(* IEC 61131-3 sources: elnaProjects/ElpcLogic/PomarKc7Unchanged/build_USO_ecl (part 3) *)

  (********************************************* Модуль A1-6 ******************************************************)

  AI_T_opornogo_podshipnika_nagnetatelia_t1_HA	:= ai.T_opornogo_podshipnika_nagnetatelia_t1.HA;
  AI_T_opornogo_podshipnika_nagnetatelia_t1_HL	:= ai.T_opornogo_podshipnika_nagnetatelia_t1.HL;
  AI_T_opornogo_podshipnika_nagnetatelia_t1_HW	:= ai.T_opornogo_podshipnika_nagnetatelia_t1.HW;
  AI_T_opornogo_podshipnika_nagnetatelia_t1_LL	:= ai.T_opornogo_podshipnika_nagnetatelia_t1.LL;
  AI_T_opornogo_podshipnika_nagnetatelia_t1_status := DWORD_TO_UDINT(ai.T_opornogo_podshipnika_nagnetatelia_t1.status);
  AI_T_opornogo_podshipnika_nagnetatelia_t1_value := ai.T_opornogo_podshipnika_nagnetatelia_t1.value;

  AI_T_opornogo_podshipnika_nagnetatelia_t2_HA	:= ai.T_opornogo_podshipnika_nagnetatelia_t2.HA;
  AI_T_opornogo_podshipnika_nagnetatelia_t2_HL	:= ai.T_opornogo_podshipnika_nagnetatelia_t2.HL;
  AI_T_opornogo_podshipnika_nagnetatelia_t2_HW	:= ai.T_opornogo_podshipnika_nagnetatelia_t2.HW;
  AI_T_opornogo_podshipnika_nagnetatelia_t2_LL	:= ai.T_opornogo_podshipnika_nagnetatelia_t2.LL;
  AI_T_opornogo_podshipnika_nagnetatelia_t2_status := DWORD_TO_UDINT(ai.T_opornogo_podshipnika_nagnetatelia_t2.status);
  AI_T_opornogo_podshipnika_nagnetatelia_t2_value := ai.T_opornogo_podshipnika_nagnetatelia_t2.value;

  AI_T_opornogo_podshipnika_nagnetatelia_t3_HA	:= ai.T_opornogo_podshipnika_nagnetatelia_t3.HA;
  AI_T_opornogo_podshipnika_nagnetatelia_t3_HL	:= ai.T_opornogo_podshipnika_nagnetatelia_t3.HL;
  AI_T_opornogo_podshipnika_nagnetatelia_t3_HW	:= ai.T_opornogo_podshipnika_nagnetatelia_t3.HW;
  AI_T_opornogo_podshipnika_nagnetatelia_t3_LL	:= ai.T_opornogo_podshipnika_nagnetatelia_t3.LL;
  AI_T_opornogo_podshipnika_nagnetatelia_t3_status := DWORD_TO_UDINT(ai.T_opornogo_podshipnika_nagnetatelia_t3.status);
  AI_T_opornogo_podshipnika_nagnetatelia_t3_value := ai.T_opornogo_podshipnika_nagnetatelia_t3.value;

  AI_T_oporno_upornogo_podshipnika_nagnetatelia_t4_HA	:= ai.T_oporno_upornogo_podshipnika_nagnetatelia_t4.HA;
  AI_T_oporno_upornogo_podshipnika_nagnetatelia_t4_HL	:= ai.T_oporno_upornogo_podshipnika_nagnetatelia_t4.HL;
  AI_T_oporno_upornogo_podshipnika_nagnetatelia_t4_HW	:= ai.T_oporno_upornogo_podshipnika_nagnetatelia_t4.HW;
  AI_T_oporno_upornogo_podshipnika_nagnetatelia_t4_LL	:= ai.T_oporno_upornogo_podshipnika_nagnetatelia_t4.LL;
  AI_T_oporno_upornogo_podshipnika_nagnetatelia_t4_status := DWORD_TO_UDINT(ai.T_oporno_upornogo_podshipnika_nagnetatelia_t4.status);
  AI_T_oporno_upornogo_podshipnika_nagnetatelia_t4_value := ai.T_oporno_upornogo_podshipnika_nagnetatelia_t4.value;

  AI_T_masla_do_AVOM_HL	:= ai.T_masla_do_AVOM.HL;
  AI_T_masla_do_AVOM_LL	:= ai.T_masla_do_AVOM.LL;
  AI_T_masla_do_AVOM_status := DWORD_TO_UDINT(ai.T_masla_do_AVOM.status);
  AI_T_masla_do_AVOM_value := ai.T_masla_do_AVOM.value;

  AI_T_masla_posle_AVOM_HL	:= ai.T_masla_posle_AVOM.HL;
  AI_T_masla_posle_AVOM_LL	:= ai.T_masla_posle_AVOM.LL;
  AI_T_masla_posle_AVOM_status := DWORD_TO_UDINT(ai.T_masla_posle_AVOM.status);
  AI_T_masla_posle_AVOM_value := ai.T_masla_posle_AVOM.value;

  AI_T_gaz_in_nagnetatelia_HL	          := ai.T_gaz_in_nagnetatelia.HL;
  AI_T_gaz_in_nagnetatelia_LL	          := ai.T_gaz_in_nagnetatelia.LL;
  AI_T_gaz_in_nagnetatelia_status := DWORD_TO_UDINT(ai.T_gaz_in_nagnetatelia.status);
  AI_T_gaz_in_nagnetatelia_value := ai.T_gaz_in_nagnetatelia.value;

  AI_T_gaz_out_nagnetatelia_HA	          := ai.T_gaz_out_nagnetatelia.HA;
  AI_T_gaz_out_nagnetatelia_HL	          := ai.T_gaz_out_nagnetatelia.HL;
  AI_T_gaz_out_nagnetatelia_HW	          := ai.T_gaz_out_nagnetatelia.HW;
  AI_T_gaz_out_nagnetatelia_LL	          := ai.T_gaz_out_nagnetatelia.LL;
  AI_T_gaz_out_nagnetatelia_status := DWORD_TO_UDINT(ai.T_gaz_out_nagnetatelia.status);
  AI_T_gaz_out_nagnetatelia_value := ai.T_gaz_out_nagnetatelia.value;

  (********************************************* Модуль A1-7 ******************************************************)

  AI_T_clodAir_dvigatelia_t1_HL	          := ai.T_clodAir_dvigatelia_t1.HL;
  AI_T_clodAir_dvigatelia_t1_LL	          := ai.T_clodAir_dvigatelia_t1.LL;
  AI_T_clodAir_dvigatelia_t1_status := DWORD_TO_UDINT(ai.T_clodAir_dvigatelia_t1.status);
  AI_T_clodAir_dvigatelia_t1_value := ai.T_clodAir_dvigatelia_t1.value;

  AI_T_hotAir_dvigatelia_t1_HL	          := ai.T_hotAir_dvigatelia_t1.HL;
  AI_T_hotAir_dvigatelia_t1_LL	          := ai.T_hotAir_dvigatelia_t1.LL;
  AI_T_hotAir_dvigatelia_t1_status := DWORD_TO_UDINT(ai.T_hotAir_dvigatelia_t1.status);
  AI_T_hotAir_dvigatelia_t1_value := ai.T_hotAir_dvigatelia_t1.value;

  (********************************************* Модуль A1-8 ******************************************************)

  AI_dPmaslo_gaz_HL	          := ai.dPmaslo_gaz.HL;
  AI_dPmaslo_gaz_LA	          := ai.dPmaslo_gaz.LA;
  AI_dPmaslo_gaz_LL	          := ai.dPmaslo_gaz.LL;
  AI_dPmaslo_gaz_LW	          := ai.dPmaslo_gaz.LW;
  AI_dPmaslo_gaz_MaxChangeUP	          := ai.dPmaslo_gaz.MaxChangeSpeed;
  AI_dPmaslo_gaz_MaxChangeDown	          := ai.dPmaslo_gaz.MaxChangeSpeedDown;
  AI_dPmaslo_gaz_status := DWORD_TO_UDINT(ai.dPmaslo_gaz.status);
  AI_dPmaslo_gaz_value := ai.dPmaslo_gaz.value;

  AI_dP_gaza_na_konfuzore_nagnetatelia_HL	          := ai.dP_gaza_na_konfuzore_nagnetatelia.HL;
  AI_dP_gaza_na_konfuzore_nagnetatelia_LL	          := ai.dP_gaza_na_konfuzore_nagnetatelia.LL;
  AI_dP_gaza_na_konfuzore_nagnetatelia_status := DWORD_TO_UDINT(ai.dP_gaza_na_konfuzore_nagnetatelia.status);
  AI_dP_gaza_na_konfuzore_nagnetatelia_value := ai.dP_gaza_na_konfuzore_nagnetatelia.value;

  AI_P_masla_uplotneniia_HL	:= ai.P_masla_uplotneniia.HL;
  AI_P_masla_uplotneniia_LL	:= ai.P_masla_uplotneniia.LL;
  AI_P_masla_uplotneniia_status := DWORD_TO_UDINT(ai.P_masla_uplotneniia.status);
  AI_P_masla_uplotneniia_value := ai.P_masla_uplotneniia.value;

  AI_P_gaza_na_vkhode_nagnetatelia_HL	:= ai.P_gaza_na_vkhode_nagnetatelia.HL;
  AI_P_gaza_na_vkhode_nagnetatelia_LL	:= ai.P_gaza_na_vkhode_nagnetatelia.LL;
  AI_P_gaza_na_vkhode_nagnetatelia_status := DWORD_TO_UDINT(ai.P_gaza_na_vkhode_nagnetatelia.status);
  AI_P_gaza_na_vkhode_nagnetatelia_value := ai.P_gaza_na_vkhode_nagnetatelia.value;

  AI_P_gaza_na_vykhode_nagnetatelia_HL	:= ai.P_gaza_na_vykhode_nagnetatelia.HL;
  AI_P_gaza_na_vykhode_nagnetatelia_LL	:= ai.P_gaza_na_vykhode_nagnetatelia.LL;
  AI_P_gaza_na_vykhode_nagnetatelia_status := DWORD_TO_UDINT(ai.P_gaza_na_vykhode_nagnetatelia.status);
  AI_P_gaza_na_vykhode_nagnetatelia_value := ai.P_gaza_na_vykhode_nagnetatelia.value;

  AI_P_masla_smazki_nizkoe_HL	          := ai.P_masla_smazki_nizkoe.HL;
  AI_P_masla_smazki_nizkoe_LA	          := ai.P_masla_smazki_nizkoe.LA;
  AI_P_masla_smazki_nizkoe_LL	          := ai.P_masla_smazki_nizkoe.LL;
  AI_P_masla_smazki_nizkoe_LW	          := ai.P_masla_smazki_nizkoe.LW;
  AI_P_masla_smazki_nizkoe_status := DWORD_TO_UDINT(ai.P_masla_smazki_nizkoe.status);
  AI_P_masla_smazki_nizkoe_value := ai.P_masla_smazki_nizkoe.value;

  AI_P_masla_smazki_srednee_posle_nasosov_HL	:= ai.P_masla_smazki_srednee_posle_nasosov.HL;
  AI_P_masla_smazki_srednee_posle_nasosov_LL	:= ai.P_masla_smazki_srednee_posle_nasosov.LL;
  AI_P_masla_smazki_srednee_posle_nasosov_LW	:= ai.P_masla_smazki_srednee_posle_nasosov.LW;
  AI_P_masla_smazki_srednee_posle_nasosov_status := DWORD_TO_UDINT(ai.P_masla_smazki_srednee_posle_nasosov.status);
  AI_P_masla_smazki_srednee_posle_nasosov_value := ai.P_masla_smazki_srednee_posle_nasosov.value;

  (********************************************* Модуль A1-9 ******************************************************)

  AI_Vibratciia_STD_t1_HA	:= ai.Vibratciia_STD_t1.HA;
  AI_Vibratciia_STD_t1_HL	:= ai.Vibratciia_STD_t1.HL;
  AI_Vibratciia_STD_t1_HW	:= ai.Vibratciia_STD_t1.HW;
  AI_Vibratciia_STD_t1_LL	:= ai.Vibratciia_STD_t1.LL;
  AI_Vibratciia_STD_t1_status := DWORD_TO_UDINT(ai.Vibratciia_STD_t1.status);
  AI_Vibratciia_STD_t1_value := ai.Vibratciia_STD_t1.value;

  AI_Vibratciia_STD_t2_HA	:= ai.Vibratciia_STD_t2.HA;
  AI_Vibratciia_STD_t2_HL	:= ai.Vibratciia_STD_t2.HL;
  AI_Vibratciia_STD_t2_HW	:= ai.Vibratciia_STD_t2.HW;
  AI_Vibratciia_STD_t2_LL	:= ai.Vibratciia_STD_t2.LL;
  AI_Vibratciia_STD_t2_status := DWORD_TO_UDINT(ai.Vibratciia_STD_t2.status);
  AI_Vibratciia_STD_t2_value := ai.Vibratciia_STD_t2.value;

  AI_Vibratciia_rotora_nagnetatelia_t1_HA	          := ai.Vibratciia_rotora_nagnetatelia_t1.HA;
  AI_Vibratciia_rotora_nagnetatelia_t1_HL	          := ai.Vibratciia_rotora_nagnetatelia_t1.HL;
  AI_Vibratciia_rotora_nagnetatelia_t1_HW	          := ai.Vibratciia_rotora_nagnetatelia_t1.HW;
  AI_Vibratciia_rotora_nagnetatelia_t1_LL	          := ai.Vibratciia_rotora_nagnetatelia_t1.LL;
  AI_Vibratciia_rotora_nagnetatelia_t1_status := DWORD_TO_UDINT(ai.Vibratciia_rotora_nagnetatelia_t1.status);
  AI_Vibratciia_rotora_nagnetatelia_t1_value := ai.Vibratciia_rotora_nagnetatelia_t1.value;

  AI_Vibratciia_rotora_nagnetatelia_t2_HA	          := ai.Vibratciia_rotora_nagnetatelia_t2.HA;
  AI_Vibratciia_rotora_nagnetatelia_t2_HL        	:= ai.Vibratciia_rotora_nagnetatelia_t2.HL;
  AI_Vibratciia_rotora_nagnetatelia_t2_HW    	:= ai.Vibratciia_rotora_nagnetatelia_t2.HW;
  AI_Vibratciia_rotora_nagnetatelia_t2_LL    	:= ai.Vibratciia_rotora_nagnetatelia_t2.LL;
  AI_Vibratciia_rotora_nagnetatelia_t2_status := DWORD_TO_UDINT(ai.Vibratciia_rotora_nagnetatelia_t2.status);
  AI_Vibratciia_rotora_nagnetatelia_t2_value := ai.Vibratciia_rotora_nagnetatelia_t2.value;

  AI_Vibratciia_rotora_nagnetatelia_t3_HA    	:= ai.Vibratciia_rotora_nagnetatelia_t3.HA;
  AI_Vibratciia_rotora_nagnetatelia_t3_HL    	:= ai.Vibratciia_rotora_nagnetatelia_t3.HL;
  AI_Vibratciia_rotora_nagnetatelia_t3_HW    	:= ai.Vibratciia_rotora_nagnetatelia_t3.HW;
  AI_Vibratciia_rotora_nagnetatelia_t3_LL    	:= ai.Vibratciia_rotora_nagnetatelia_t3.LL;
  AI_Vibratciia_rotora_nagnetatelia_t3_status := DWORD_TO_UDINT(ai.Vibratciia_rotora_nagnetatelia_t3.status);
  AI_Vibratciia_rotora_nagnetatelia_t3_value := ai.Vibratciia_rotora_nagnetatelia_t3.value;

  AI_Vibratciia_rotora_nagnetatelia_t4_HA    	:= ai.Vibratciia_rotora_nagnetatelia_t4.HA;
  AI_Vibratciia_rotora_nagnetatelia_t4_HL    	:= ai.Vibratciia_rotora_nagnetatelia_t4.HL;
  AI_Vibratciia_rotora_nagnetatelia_t4_HW    	:= ai.Vibratciia_rotora_nagnetatelia_t4.HW;
  AI_Vibratciia_rotora_nagnetatelia_t4_LL    	:= ai.Vibratciia_rotora_nagnetatelia_t4.LL;
  AI_Vibratciia_rotora_nagnetatelia_t4_status := DWORD_TO_UDINT(ai.Vibratciia_rotora_nagnetatelia_t4.status);
  AI_Vibratciia_rotora_nagnetatelia_t4_value := ai.Vibratciia_rotora_nagnetatelia_t4.value;

  AI_Osevoi_sdvig_rotora_nagnetatelia_HA    	:= ai.Osevoi_sdvig_rotora_nagnetatelia.HA;
  AI_Osevoi_sdvig_rotora_nagnetatelia_HL    	:= ai.Osevoi_sdvig_rotora_nagnetatelia.HL;
  AI_Osevoi_sdvig_rotora_nagnetatelia_HW    	:= ai.Osevoi_sdvig_rotora_nagnetatelia.HW;
  AI_Osevoi_sdvig_rotora_nagnetatelia_LA    	:= ai.Osevoi_sdvig_rotora_nagnetatelia.LA;
  AI_Osevoi_sdvig_rotora_nagnetatelia_LL    	:= ai.Osevoi_sdvig_rotora_nagnetatelia.LL;
  AI_Osevoi_sdvig_rotora_nagnetatelia_LW    	:= ai.Osevoi_sdvig_rotora_nagnetatelia.LW;
  AI_Osevoi_sdvig_rotora_nagnetatelia_status := DWORD_TO_UDINT(ai.Osevoi_sdvig_rotora_nagnetatelia.status);
  AI_Osevoi_sdvig_rotora_nagnetatelia_value := ai.Osevoi_sdvig_rotora_nagnetatelia.value;

  AI_Uroven_masla_v_maslobake_HL	:= ai.Uroven_masla_v_maslobake.HL;
  AI_Uroven_masla_v_maslobake_HW	:= ai.Uroven_masla_v_maslobake.HW;
  AI_Uroven_masla_v_maslobake_LA	:= ai.Uroven_masla_v_maslobake.LA;
  AI_Uroven_masla_v_maslobake_LL	:= ai.Uroven_masla_v_maslobake.LL;
  AI_Uroven_masla_v_maslobake_LW	:= ai.Uroven_masla_v_maslobake.LW;
  AI_Uroven_masla_v_maslobake_status := DWORD_TO_UDINT(ai.Uroven_masla_v_maslobake.status);
  AI_Uroven_masla_v_maslobake_value := ai.Uroven_masla_v_maslobake.value;

  (********************************************* Модуль A1-10 ******************************************************)

  AI_T_vnytri_shkafa_HL	:= ai.T_vnytri_shkafa.HL;
  AI_T_vnytri_shkafa_LL	:= ai.T_vnytri_shkafa.LL;
  AI_T_vnytri_shkafa_HW	:= ai.T_vnytri_shkafa.HL;
  AI_T_vnytri_shkafa_LW	:= ai.T_vnytri_shkafa.LL;
  AI_T_vnytri_shkafa_status     := DWORD_TO_UDINT(ai.T_vnytri_shkafa.status);
  AI_T_vnytri_shkafa_value      := ai.T_vnytri_shkafa.value;

  AI_Tok_vozbuzhdeniia_vozbuditelia_HL	:= ai.Tok_vozbuzhdeniia_vozbuditelia.HL;
  AI_Tok_vozbuzhdeniia_vozbuditelia_LL	:= ai.Tok_vozbuzhdeniia_vozbuditelia.LL;
  AI_Tok_vozbuzhdeniia_vozbuditelia_status := DWORD_TO_UDINT(ai.Tok_vozbuzhdeniia_vozbuditelia.status);
  AI_Tok_vozbuzhdeniia_vozbuditelia_value := ai.Tok_vozbuzhdeniia_vozbuditelia.value;

  AI_Tok_statora_elektrodvigatelia_HL	:= ai.Tok_statora_elektrodvigatelia.HL;
  AI_Tok_statora_elektrodvigatelia_LL	:= ai.Tok_statora_elektrodvigatelia.LL;
  AI_Tok_statora_elektrodvigatelia_status := DWORD_TO_UDINT(ai.Tok_statora_elektrodvigatelia.status);
  AI_Tok_statora_elektrodvigatelia_value := ai.Tok_statora_elektrodvigatelia.value;

  AI_Aktivnaia_moshchnost_HL	:= ai.Aktivnaia_moshchnost.HL;
  AI_Aktivnaia_moshchnost_LL	:= ai.Aktivnaia_moshchnost.LL;
  AI_Aktivnaia_moshchnost_status := DWORD_TO_UDINT(ai.Aktivnaia_moshchnost.status);
  AI_Aktivnaia_moshchnost_value := ai.Aktivnaia_moshchnost.value;

  AI_Reaktivnaia_moshchnost_HL    	:= ai.Reaktivnaia_moshchnost.HL;
  AI_Reaktivnaia_moshchnost_LL    	:= ai.Reaktivnaia_moshchnost.LL;
  AI_Reaktivnaia_moshchnost_status := DWORD_TO_UDINT(ai.Reaktivnaia_moshchnost.status);
  AI_Reaktivnaia_moshchnost_value := ai.Reaktivnaia_moshchnost.value;

  AI_VoltageSHU_osnovnoi_vvod_HL	:= ai.VoltageSHU_osnovnoi_vvod.HL;
  AI_VoltageSHU_osnovnoi_vvod_HW	:= ai.VoltageSHU_osnovnoi_vvod.HW;
  AI_VoltageSHU_osnovnoi_vvod_LL	:= ai.VoltageSHU_osnovnoi_vvod.LL;
  AI_VoltageSHU_osnovnoi_vvod_LW	:= ai.VoltageSHU_osnovnoi_vvod.LW;
  AI_VoltageSHU_osnovnoi_vvod_status := DWORD_TO_UDINT(ai.VoltageSHU_osnovnoi_vvod.status);
  AI_VoltageSHU_osnovnoi_vvod_value := ai.VoltageSHU_osnovnoi_vvod.value;

  AI_VoltageSHU_rezervnyi_vvod_HL	:= ai.VoltageSHU_rezervnyi_vvod.HL;
  AI_VoltageSHU_rezervnyi_vvod_HW	:= ai.VoltageSHU_rezervnyi_vvod.HW;
  AI_VoltageSHU_rezervnyi_vvod_LL	:= ai.VoltageSHU_rezervnyi_vvod.LL;
  AI_VoltageSHU_rezervnyi_vvod_LW	:= ai.VoltageSHU_rezervnyi_vvod.LW;
  AI_VoltageSHU_rezervnyi_vvod_status := DWORD_TO_UDINT(ai.VoltageSHU_rezervnyi_vvod.status);
  AI_VoltageSHU_rezervnyi_vvod_value := ai.VoltageSHU_rezervnyi_vvod.value;

  algoritms_AntiPompag_q_status	          := DWORD_TO_UDINT(ai.Rashod.status);
  algoritms_AntiPompag_q_Value	          := ai.Rashod.value;
  algoritms_AntiPompag_zapas_status	:= DWORD_TO_UDINT(ai.Zapas.status);
  algoritms_AntiPompag_zapas_Value	:= ai.Zapas.value;
END_FUNCTION_BLOCK

FUNCTION_BLOCK OPC_protections_get
  VAR_EXTERNAL
    protections : ProtectionsConfig;
    protections_AO_KC_inCommand_ARM : UINT;
    protections_AO_PRU_inCommand_ARM : UINT;
    protections_AO_SHU_inCommand_ARM : UINT;
    protections_BEAO_knSHU_inCommand_ARM : UINT;
    protections_DavlenieMaslaSmazkiDi_inCommand_ARM : UINT;
    protections_EAO_PRU_inCommand_ARM : UINT;
    protections_Kran1sdvig_inCommand_ARM : UINT;
    protections_Kran2sdvig_inCommand_ARM : UINT;
    protections_Osevoi_sdvig_rotora_nagnetatelia_HA_inCommand_ARM : UINT;
    protections_OsevojSdvigLevyjDi_inCommand_ARM : UINT;
    protections_OsevojSdvigPravyjDi_inCommand_ARM : UINT;
    protections_P_masla_smazki_nizkoe_LA_inCommand_ARM : UINT;
    protections_Srab_BEAO_inCommand_ARM : UINT;
    protections_T_gaza_na_vykhode_nagnetatelia_HA_inCommand_ARM : UINT;
    protections_T_opornogo_podshipnika_nagnetatelia_t1_HA_inCommand_ARM : UINT;
    protections_T_opornogo_podshipnika_nagnetatelia_t2_HA_inCommand_ARM : UINT;
    protections_T_opornogo_podshipnika_nagnetatelia_t3_HA_inCommand_ARM : UINT;
    protections_T_opornoupornogo_podshipnika_nagnetatelia_t4_HA_inCommand_ARM : UINT;
    protections_T_perednego_opornogo_podshipnika_dvigatelia_t1_HA_inCommand_ARM : UINT;
    protections_T_podshipnika_reduktora_t1_HA_inCommand_ARM : UINT;
    protections_T_podshipnika_reduktora_t2_HA_inCommand_ARM : UINT;
    protections_T_podshipnika_reduktora_t3_HA_inCommand_ARM : UINT;
    protections_T_podshipnika_reduktora_t4_HA_inCommand_ARM : UINT;
    protections_T_zadnego_opornogo_podshipnika_dvigatelia_t2_HA_inCommand_ARM : UINT;
    protections_Uroven_masla_v_maslobake_LA_inCommand_ARM : UINT;
    protections_Vibratciia_STD_t1_HA_inCommand_ARM : UINT;
    protections_Vibratciia_STD_t2_HA_inCommand_ARM : UINT;
    protections_Vibratciia_rotora_nagnetatelia_t1_HA_inCommand_ARM : UINT;
    protections_Vibratciia_rotora_nagnetatelia_t2_HA_inCommand_ARM : UINT;
    protections_Vibratciia_rotora_nagnetatelia_t3_HA_inCommand_ARM : UINT;
    protections_Vibratciia_rotora_nagnetatelia_t4_HA_inCommand_ARM : UINT;
    protections_dP_masloGaz_LowDI_inCommand_ARM : UINT;
    protections_dP_maslogaz_LA_inCommand_ARM : UINT;
    protections_mvOff_inCommand_ARM : UINT;
  END_VAR

  (* OPC Get - IM. Чтение текущих состояний тэгов _______________________________________________________*)

  protections.AO_KC.inCommand_ARM	:= UINT_TO_WORD(protections_AO_KC_inCommand_ARM);
  protections.AO_PRU.inCommand_ARM	:= UINT_TO_WORD(protections_AO_PRU_inCommand_ARM);
  protections.AO_SHU.inCommand_ARM	:= UINT_TO_WORD(protections_AO_SHU_inCommand_ARM);
  protections.BEAO_knSHU.inCommand_ARM	:= UINT_TO_WORD(protections_BEAO_knSHU_inCommand_ARM);
  protections.DavlenieMaslaSmazkiDi.inCommand_ARM	:= UINT_TO_WORD(protections_DavlenieMaslaSmazkiDi_inCommand_ARM);
  protections.dP_maslogaz_LA.inCommand_ARM	:= UINT_TO_WORD(protections_dP_maslogaz_LA_inCommand_ARM);
  protections.dP_masloGaz_LowDI.inCommand_ARM	:= UINT_TO_WORD(protections_dP_masloGaz_LowDI_inCommand_ARM);
  protections.EAO_PRU.inCommand_ARM	:= UINT_TO_WORD(protections_EAO_PRU_inCommand_ARM);
  protections.mvOff.inCommand_ARM	:= UINT_TO_WORD(protections_mvOff_inCommand_ARM);
  protections.Osevoi_sdvig_rotora_nagnetatelia_HA.inCommand_ARM	:= UINT_TO_WORD(protections_Osevoi_sdvig_rotora_nagnetatelia_HA_inCommand_ARM);
  protections.OsevojSdvigLevyjDi.inCommand_ARM	:= UINT_TO_WORD(protections_OsevojSdvigLevyjDi_inCommand_ARM);
  protections.OsevojSdvigPravyjDi.inCommand_ARM	:= UINT_TO_WORD(protections_OsevojSdvigPravyjDi_inCommand_ARM);
  protections.Srab_BEAO.inCommand_ARM	:= UINT_TO_WORD(protections_Srab_BEAO_inCommand_ARM);
  protections.T_gaza_na_vykhode_nagnetatelia_HA.inCommand_ARM	:= UINT_TO_WORD(protections_T_gaza_na_vykhode_nagnetatelia_HA_inCommand_ARM);
  protections.T_opornogo_podshipnika_nagnetatelia_t1_HA.inCommand_ARM	:= UINT_TO_WORD(protections_T_opornogo_podshipnika_nagnetatelia_t1_HA_inCommand_ARM);
  protections.T_opornogo_podshipnika_nagnetatelia_t2_HA.inCommand_ARM	:= UINT_TO_WORD(protections_T_opornogo_podshipnika_nagnetatelia_t2_HA_inCommand_ARM);
  protections.T_opornogo_podshipnika_nagnetatelia_t3_HA.inCommand_ARM	:= UINT_TO_WORD(protections_T_opornogo_podshipnika_nagnetatelia_t3_HA_inCommand_ARM);
  protections.T_opornoupornogo_podshipnika_nagnetatelia_t4_HA.inCommand_ARM	:= UINT_TO_WORD(protections_T_opornoupornogo_podshipnika_nagnetatelia_t4_HA_inCommand_ARM);
  protections.T_perednego_opornogo_podshipnika_dvigatelia_t1_HA.inCommand_ARM	:= UINT_TO_WORD(protections_T_perednego_opornogo_podshipnika_dvigatelia_t1_HA_inCommand_ARM);
  protections.T_podshipnika_reduktora_t1_HA.inCommand_ARM	:= UINT_TO_WORD(protections_T_podshipnika_reduktora_t1_HA_inCommand_ARM);
  protections.T_podshipnika_reduktora_t2_HA.inCommand_ARM	:= UINT_TO_WORD(protections_T_podshipnika_reduktora_t2_HA_inCommand_ARM);
  protections.T_podshipnika_reduktora_t3_HA.inCommand_ARM	:= UINT_TO_WORD(protections_T_podshipnika_reduktora_t3_HA_inCommand_ARM);
  protections.T_podshipnika_reduktora_t4_HA.inCommand_ARM	:= UINT_TO_WORD(protections_T_podshipnika_reduktora_t4_HA_inCommand_ARM);
  protections.T_zadnego_opornogo_podshipnika_dvigatelia_t2_HA.inCommand_ARM	:= UINT_TO_WORD(protections_T_zadnego_opornogo_podshipnika_dvigatelia_t2_HA_inCommand_ARM);
  protections.Uroven_masla_v_maslobake_LA.inCommand_ARM	:= UINT_TO_WORD(protections_Uroven_masla_v_maslobake_LA_inCommand_ARM);
  protections.Vibratciia_rotora_nagnetatelia_t1_HA.inCommand_ARM	:= UINT_TO_WORD(protections_Vibratciia_rotora_nagnetatelia_t1_HA_inCommand_ARM);
  protections.Vibratciia_rotora_nagnetatelia_t2_HA.inCommand_ARM	:= UINT_TO_WORD(protections_Vibratciia_rotora_nagnetatelia_t2_HA_inCommand_ARM);
  protections.Vibratciia_rotora_nagnetatelia_t3_HA.inCommand_ARM	:= UINT_TO_WORD(protections_Vibratciia_rotora_nagnetatelia_t3_HA_inCommand_ARM);
  protections.Vibratciia_rotora_nagnetatelia_t4_HA.inCommand_ARM	:= UINT_TO_WORD(protections_Vibratciia_rotora_nagnetatelia_t4_HA_inCommand_ARM);
  protections.Vibratciia_STD_t1_HA.inCommand_ARM	:= UINT_TO_WORD(protections_Vibratciia_STD_t1_HA_inCommand_ARM);
  protections.Vibratciia_STD_t2_HA.inCommand_ARM	:= UINT_TO_WORD(protections_Vibratciia_STD_t2_HA_inCommand_ARM);
  protections.Kran1sdvig.inCommand_ARM	:= UINT_TO_WORD(protections_Kran1sdvig_inCommand_ARM);
  protections.Kran2sdvig.inCommand_ARM	:= UINT_TO_WORD(protections_Kran2sdvig_inCommand_ARM);
  protections.P_masla_smazki_nizkoe_LA.inCommand_ARM	:= UINT_TO_WORD(protections_P_masla_smazki_nizkoe_LA_inCommand_ARM);
END_FUNCTION_BLOCK

FUNCTION_BLOCK OPC_protections_set
  VAR_EXTERNAL
    protections_AO_KC_status : UDINT;
    protections_AO_PRU_status : UDINT;
    protections_AO_SHU_status : UDINT;
    protections_BEAO_knSHU_status : UDINT;
    protections_DavlenieMaslaSmazkiDi_status : UDINT;
    protections_EAO_PRU_status : UDINT;
    protections_Kran1sdvig_status : UDINT;
    protections_Kran2sdvig_status : UDINT;
    protections_Osevoi_sdvig_rotora_nagnetatelia_HA_status : UDINT;
    protections_OsevojSdvigLevyjDi_status : UDINT;
    protections_OsevojSdvigPravyjDi_status : UDINT;
    protections_P_masla_smazki_nizkoe_LA_status : UDINT;
    protections_Srab_BEAO_status : UDINT;
    protections_T_gaza_na_vykhode_nagnetatelia_HA_status : UDINT;
    protections_T_opornogo_podshipnika_nagnetatelia_t1_HA_status : UDINT;
    protections_T_opornogo_podshipnika_nagnetatelia_t2_HA_status : UDINT;
    protections_T_opornogo_podshipnika_nagnetatelia_t3_HA_status : UDINT;
    protections_T_opornoupornogo_podshipnika_nagnetatelia_t4_HA_status : UDINT;
    protections_T_perednego_opornogo_podshipnika_dvigatelia_t1_HA_status : UDINT;
    protections_T_podshipnika_reduktora_t1_HA_status : UDINT;
    protections_T_podshipnika_reduktora_t2_HA_status : UDINT;
    protections_T_podshipnika_reduktora_t3_HA_status : UDINT;
    protections_T_podshipnika_reduktora_t4_HA_status : UDINT;
    protections_T_zadnego_opornogo_podshipnika_dvigatelia_t2_HA_status : UDINT;
    protections_Uroven_masla_v_maslobake_LA_status : UDINT;
    protections_Vibratciia_STD_t1_HA_status : UDINT;
    protections_Vibratciia_STD_t2_HA_status : UDINT;
    protections_Vibratciia_rotora_nagnetatelia_t1_HA_status : UDINT;
    protections_Vibratciia_rotora_nagnetatelia_t2_HA_status : UDINT;
    protections_Vibratciia_rotora_nagnetatelia_t3_HA_status : UDINT;
    protections_Vibratciia_rotora_nagnetatelia_t4_HA_status : UDINT;
    protections_dP_masloGaz_LowDI_status : UDINT;
    protections_dP_maslogaz_LA_status : UDINT;
    protections_mvOff_status : UDINT;
    protections : ProtectionsConfig;
  END_VAR

  (* OPC Set - IM. Запись текущих состояний тэгов _______________________________________________________*)

  protections_AO_KC_status	:= DWORD_TO_UDINT(protections.AO_KC.status);
  protections_AO_PRU_status	:= DWORD_TO_UDINT(protections.AO_PRU.status);
  protections_AO_SHU_status	:= DWORD_TO_UDINT(protections.AO_SHU.status);
  protections_BEAO_knSHU_status	:= DWORD_TO_UDINT(protections.BEAO_knSHU.status);
  protections_DavlenieMaslaSmazkiDi_status	:= DWORD_TO_UDINT(protections.DavlenieMaslaSmazkiDi.status);
  protections_P_masla_smazki_nizkoe_LA_status	:= DWORD_TO_UDINT(protections.P_masla_smazki_nizkoe_LA.status);
  protections_dP_maslogaz_LA_status	:= DWORD_TO_UDINT(protections.dP_maslogaz_LA.status);
  protections_dP_masloGaz_LowDI_status	:= DWORD_TO_UDINT(protections.dP_masloGaz_LowDI.status);
  protections_EAO_PRU_status	:= DWORD_TO_UDINT(protections.EAO_PRU.status);
  protections_mvOff_status	:= DWORD_TO_UDINT(protections.mvOff.status);
  protections_OsevojSdvigLevyjDi_status	:= DWORD_TO_UDINT(protections.OsevojSdvigLevyjDi.status);
  protections_OsevojSdvigPravyjDi_status	:= DWORD_TO_UDINT(protections.OsevojSdvigPravyjDi.status);
  protections_Osevoi_sdvig_rotora_nagnetatelia_HA_status	:= DWORD_TO_UDINT(protections.Osevoi_sdvig_rotora_nagnetatelia_HA.status);
  protections_T_gaza_na_vykhode_nagnetatelia_HA_status	:= DWORD_TO_UDINT(protections.T_gaza_na_vykhode_nagnetatelia_HA.status);
  protections_Srab_BEAO_status	:= DWORD_TO_UDINT(protections.Srab_BEAO.status);
  protections_T_opornogo_podshipnika_nagnetatelia_t1_HA_status	:= DWORD_TO_UDINT(protections.T_opornogo_podshipnika_nagnetatelia_t1_HA.status);
  protections_T_opornogo_podshipnika_nagnetatelia_t2_HA_status	:= DWORD_TO_UDINT(protections.T_opornogo_podshipnika_nagnetatelia_t2_HA.status);
  protections_T_opornogo_podshipnika_nagnetatelia_t3_HA_status	:= DWORD_TO_UDINT(protections.T_opornogo_podshipnika_nagnetatelia_t3_HA.status);
  protections_T_opornoupornogo_podshipnika_nagnetatelia_t4_HA_status	:= DWORD_TO_UDINT(protections.T_opornoupornogo_podshipnika_nagnetatelia_t4_HA.status);
  protections_T_perednego_opornogo_podshipnika_dvigatelia_t1_HA_status	:= DWORD_TO_UDINT(protections.T_perednego_opornogo_podshipnika_dvigatelia_t1_HA.status);
  protections_T_zadnego_opornogo_podshipnika_dvigatelia_t2_HA_status	:= DWORD_TO_UDINT(protections.T_zadnego_opornogo_podshipnika_dvigatelia_t2_HA.status);
  protections_T_podshipnika_reduktora_t1_HA_status	:= DWORD_TO_UDINT(protections.T_podshipnika_reduktora_t1_HA.status);
  protections_T_podshipnika_reduktora_t2_HA_status	:= DWORD_TO_UDINT(protections.T_podshipnika_reduktora_t2_HA.status);
  protections_T_podshipnika_reduktora_t3_HA_status	:= DWORD_TO_UDINT(protections.T_podshipnika_reduktora_t3_HA.status);
  protections_T_podshipnika_reduktora_t4_HA_status	:= DWORD_TO_UDINT(protections.T_podshipnika_reduktora_t4_HA.status);
  protections_Uroven_masla_v_maslobake_LA_status	:= DWORD_TO_UDINT(protections.Uroven_masla_v_maslobake_LA.status);
  protections_Vibratciia_rotora_nagnetatelia_t1_HA_status	:= DWORD_TO_UDINT(protections.Vibratciia_rotora_nagnetatelia_t1_HA.status);
  protections_Vibratciia_rotora_nagnetatelia_t2_HA_status	:= DWORD_TO_UDINT(protections.Vibratciia_rotora_nagnetatelia_t2_HA.status);
  protections_Vibratciia_rotora_nagnetatelia_t3_HA_status	:= DWORD_TO_UDINT(protections.Vibratciia_rotora_nagnetatelia_t3_HA.status);
  protections_Vibratciia_rotora_nagnetatelia_t4_HA_status	:= DWORD_TO_UDINT(protections.Vibratciia_rotora_nagnetatelia_t4_HA.status);
  protections_Vibratciia_STD_t1_HA_status	:= DWORD_TO_UDINT(protections.Vibratciia_STD_t1_HA.status);
  protections_Vibratciia_STD_t2_HA_status	:= DWORD_TO_UDINT(protections.Vibratciia_STD_t2_HA.status);
  protections_Kran1sdvig_status	:= DWORD_TO_UDINT(protections.Kran1sdvig.status);
  protections_Kran2sdvig_status	:= DWORD_TO_UDINT(protections.Kran2sdvig.status);
END_FUNCTION_BLOCK

FUNCTION_BLOCK OPC_algoritms_set
  VAR_EXTERNAL
    algoritms : AlgoritmsConfig;
    algManager_Mode : UINT;
    algoritms_AutoAvom_status : UDINT;
    algoritms_AutoPns_OffTimer : UINT;
    algoritms_AutoPns_OnTimer : UINT;
    algoritms_AutoPns_status : UDINT;
    algoritms_AutoTen_status : UDINT;
    algoritms_Remont_status : UDINT;
    algoritms_TestProtection_status : UDINT;
    algoritms_autoNu_NotHasRezervNU : BOOL;
    algoritms_autoNu_status : UDINT;
    algoritms_puskOilSystem_Error : UDINT;
    algoritms_puskOilSystem_Start : UDINT;
    algoritms_puskOilSystem_Top : UDINT;
    algoritms_puskOilSystem_status : UDINT;
    algoritms_testIm_status : UDINT;
    algoritms_vibegPNS_Error : UDINT;
    algoritms_vibegPNS_Start : UDINT;
    algoritms_vibegPNS_Top : UDINT;
    algoritms_vibegPNS_algContinue_status : UDINT;
    algoritms_vibegPNS_status : UDINT;
    algoritms_vibegPNS_waitVibeg_timer : UINT;
    protectManager_protectionInRemont : BOOL;
    algManager : struct_AlgoritmsManager;
    protectManager : struct_ProtectionsManager;
    NotHasRezervNU : BOOL;
    AlgTimers : struct_AlgTimers;
    AlgQuestions : AlgoritmsQuestions;
    algoritms_Apusk_Error : UDINT;
    algoritms_Apusk_Start : UDINT;
    algoritms_Apusk_Top : UDINT;
    algoritms_Apusk_status : UDINT;
    algoritms_RingToLine_Error : UDINT;
    algoritms_RingToLine_Start : UDINT;
    algoritms_RingToLine_Top : UDINT;
    algoritms_RingToLine_status : UDINT;
    algoritms_SemiAutoPusk_Error : UDINT;
    algoritms_SemiAutoPusk_Start : UDINT;
    algoritms_SemiAutoPusk_Top : UDINT;
    algoritms_SemiAutoPusk_cmdRun1ph_status : UDINT;
    algoritms_SemiAutoPusk_cmdRun2ph_status : UDINT;
    algoritms_SemiAutoPusk_cmdRun3ph_status : UDINT;
    algoritms_SemiAutoPusk_cmdRun4ph_status : UDINT;
    algoritms_SemiAutoPusk_status : UDINT;
    algoritms_ao_Error : UDINT;
    algoritms_ao_Start : UDINT;
    algoritms_ao_Top : UDINT;
    algoritms_ao_status : UDINT;
    algoritms_ao_waitKran_timer : UINT;
    algoritms_engineRun_BreakPuskTimer_timer : UINT;
    algoritms_engineRun_Error : UDINT;
    algoritms_engineRun_Start : UDINT;
    algoritms_engineRun_Top : UDINT;
    algoritms_engineRun_status : UDINT;
    algoritms_filling_BreakPuskTimer_timer : UINT;
    algoritms_filling_Error : UDINT;
    algoritms_filling_Start : UDINT;
    algoritms_filling_Top : UDINT;
    algoritms_filling_status : UDINT;
    algoritms_filling_waitAfterKran4_timer : UINT;
    algoritms_filling_waitAfterKran5_timer : UINT;
    algoritms_no_Error : UDINT;
    algoritms_no_Start : UDINT;
    algoritms_no_Top : UDINT;
    algoritms_no_status : UDINT;
    algoritms_no_waitCloseKran_timer : UINT;
    algoritms_ppu_Error : UDINT;
    algoritms_ppu_Start : UDINT;
    algoritms_ppu_Top : UDINT;
    algoritms_ppu_status : UDINT;
    algoritms_puskK_Error : UDINT;
    algoritms_puskK_Start : UDINT;
    algoritms_puskK_Top : UDINT;
    algoritms_puskK_questionFilling_status : UDINT;
    algoritms_puskK_questionUnload_status : UDINT;
    algoritms_puskK_status : UDINT;
    algoritms_puskK_wait720_timer : UINT;
    algoritms_puskOilSystem_BreakPuskTimer_Poil_timer : UINT;
    algoritms_puskOilSystem_BreakPuskTimer_dPmg_timer : UINT;
    algoritms_puskV_Error : UDINT;
    algoritms_puskV_Start : UDINT;
    algoritms_puskV_Top : UDINT;
    algoritms_puskV_questionFilling_status : UDINT;
    algoritms_puskV_questionMVoff_status : UDINT;
    algoritms_puskV_status : UDINT;
    algoritms_puskV_wait600_timer : UINT;
    algoritms_testPms_BreakTest_timer : UINT;
    algoritms_testPms_Error : UDINT;
    algoritms_testPms_Start : UDINT;
    algoritms_testPms_Top : UDINT;
    algoritms_testPms_algContinue_status : UDINT;
    algoritms_testPms_status : UDINT;
    algoritms_testdPmg_BreakTest_timer : UINT;
    algoritms_testdPmg_Error : UDINT;
    algoritms_testdPmg_Start : UDINT;
    algoritms_testdPmg_Top : UDINT;
    algoritms_testdPmg_algContinue_status : UDINT;
    algoritms_testdPmg_status : UDINT;
  END_VAR

  (* OPC Set - algoritms. Запись текущих состояний тэгов _______________________________________________________*)

  algManager_Mode := algManager.mode;

  protectManager_protectionInRemont:= protectManager.protectionInRemont;

  algoritms_autoNu_NotHasRezervNU:= NotHasRezervNU;

  algoritms_no_Start	:= DWORD_TO_UDINT(algoritms.no.Start);
  algoritms_no_Error	:= DWORD_TO_UDINT(algoritms.no.Error);
  algoritms_no_Top	:= DWORD_TO_UDINT(algoritms.no.Top);
  algoritms_no_status	:= DWORD_TO_UDINT(algoritms.no.status);
  algoritms_no_waitCloseKran_timer	:= AlgTimers.NO_waitCloseKran;

  algoritms_ao_Start	:= DWORD_TO_UDINT(algoritms.ao.Start);
  algoritms_ao_Error	:= DWORD_TO_UDINT(algoritms.ao.Error);
  algoritms_ao_Top	:= DWORD_TO_UDINT(algoritms.ao.Top);
  algoritms_ao_status	:= DWORD_TO_UDINT(algoritms.ao.status);
  algoritms_ao_waitKran_timer	:= AlgTimers.AO_waitKran;

  algoritms_vibegPNS_Start		:= DWORD_TO_UDINT(algoritms.vibegPNS.Start);
  algoritms_vibegPNS_Error		:= DWORD_TO_UDINT(algoritms.vibegPNS.Error);
  algoritms_vibegPNS_Top		:= DWORD_TO_UDINT(algoritms.vibegPNS.Top);
  algoritms_vibegPNS_status		:= DWORD_TO_UDINT(algoritms.vibegPNS.status);
  algoritms_vibegPNS_waitVibeg_timer	:= AlgTimers.vibegPNS_Timer;
  algoritms_vibegPNS_algContinue_status	:= DWORD_TO_UDINT(AlgQuestions.vibegPNS_algContinue.status);

  algoritms_testPms_Start		:= DWORD_TO_UDINT(algoritms.testPms.Start);
  algoritms_testPms_Error		:= DWORD_TO_UDINT(algoritms.testPms.Error);
  algoritms_testPms_Top		:= DWORD_TO_UDINT(algoritms.testPms.Top);
  algoritms_testPms_status		:= DWORD_TO_UDINT(algoritms.testPms.status);
  algoritms_testPms_algContinue_status	:= DWORD_TO_UDINT(AlgQuestions.testPms_algContinue.status);
  algoritms_testPms_BreakTest_timer	:= AlgTimers.testPms_BreakTest;

  algoritms_testdPmg_Start		:= DWORD_TO_UDINT(algoritms.testdPmg.Start);
  algoritms_testdPmg_Error		:= DWORD_TO_UDINT(algoritms.testdPmg.Error);
  algoritms_testdPmg_Top		:= DWORD_TO_UDINT(algoritms.testdPmg.Top);
  algoritms_testdPmg_status		:= DWORD_TO_UDINT(algoritms.testdPmg.status);
  algoritms_testdPmg_algContinue_status	:= DWORD_TO_UDINT(AlgQuestions.testdPmg_algContinue.status);
  algoritms_testdPmg_BreakTest_timer	:= AlgTimers.testdPmg_BreakTest;

  algoritms_testIm_status	:= DWORD_TO_UDINT(algoritms.testIm.status);

  algoritms_ppu_status	:= DWORD_TO_UDINT(algoritms.ppu.status);
  algoritms_ppu_Start	          := DWORD_TO_UDINT(algoritms.ppu.Start);
  algoritms_ppu_Error	          := DWORD_TO_UDINT(algoritms.ppu.Error);
  algoritms_ppu_Top	          := DWORD_TO_UDINT(algoritms.ppu.Top);

  algoritms_puskOilSystem_status			:= DWORD_TO_UDINT(algoritms.puskOilSystem.status);
  algoritms_puskOilSystem_Start				:= DWORD_TO_UDINT(algoritms.puskOilSystem.Start);
  algoritms_puskOilSystem_Error				:= DWORD_TO_UDINT(algoritms.puskOilSystem.Error);
  algoritms_puskOilSystem_Top				:= DWORD_TO_UDINT(algoritms.puskOilSystem.Top);
  algoritms_puskOilSystem_BreakPuskTimer_Poil_timer	          := AlgTimers.puskOilSystem_BreakPuskTimer_Poil;

  algoritms_engineRun_status			:= DWORD_TO_UDINT(algoritms.engineRun.status);
  algoritms_engineRun_Start			:= DWORD_TO_UDINT(algoritms.engineRun.Start);
  algoritms_engineRun_Error			:= DWORD_TO_UDINT(algoritms.engineRun.Error);
  algoritms_engineRun_Top			:= DWORD_TO_UDINT(algoritms.engineRun.Top);
  algoritms_engineRun_BreakPuskTimer_timer	:= AlgTimers.engineRun_BreakPuskTimer;

  algoritms_filling_status		:= DWORD_TO_UDINT(algoritms.filling.status);
  algoritms_filling_Start		:= DWORD_TO_UDINT(algoritms.filling.Start);
  algoritms_filling_Error		:= DWORD_TO_UDINT(algoritms.filling.Error);
  algoritms_filling_Top		:= DWORD_TO_UDINT(algoritms.filling.Top);
  algoritms_filling_BreakPuskTimer_timer	:= AlgTimers.filling_BreakPuskTimer;
  algoritms_filling_waitAfterKran4_timer	:= AlgTimers.filling_waitAfterKran4;
  algoritms_filling_waitAfterKran5_timer	:= AlgTimers.filling_waitAfterKran5;

  algoritms_RingToLine_status	:= DWORD_TO_UDINT(algoritms.RingToLine.status);
  algoritms_RingToLine_Start	:= DWORD_TO_UDINT(algoritms.RingToLine.Start);
  algoritms_RingToLine_Error	:= DWORD_TO_UDINT(algoritms.RingToLine.Error);
  algoritms_RingToLine_Top	:= DWORD_TO_UDINT(algoritms.RingToLine.Top);

  algoritms_puskK_status	            := DWORD_TO_UDINT(algoritms.puskK.status);
  algoritms_puskK_Start	            := DWORD_TO_UDINT(algoritms.puskK.Start);
  algoritms_puskK_Error	            := DWORD_TO_UDINT(algoritms.puskK.Error);
  algoritms_puskK_Top	                      := DWORD_TO_UDINT(algoritms.puskK.Top);
  algoritms_puskK_wait720_timer	            := AlgTimers.puskK_wait720;
  algoritms_puskK_questionFilling_status	  := DWORD_TO_UDINT(AlgQuestions.puskK_questionFilling.status);
  algoritms_puskK_questionUnload_status	  := DWORD_TO_UDINT(AlgQuestions.puskK_questionUnload.status);

  algoritms_puskV_status	          := DWORD_TO_UDINT(algoritms.puskV.status);
  algoritms_puskV_Start	          := DWORD_TO_UDINT(algoritms.puskV.Start);
  algoritms_puskV_Error	          := DWORD_TO_UDINT(algoritms.puskV.Error);
  algoritms_puskV_Top	                    := DWORD_TO_UDINT(algoritms.puskV.Top);
  algoritms_puskV_wait600_timer	          := AlgTimers.puskV_wait600;
  algoritms_puskV_questionFilling_status	:= DWORD_TO_UDINT(AlgQuestions.puskV_questionEngine.status);
  algoritms_puskV_questionMVoff_status	:= DWORD_TO_UDINT(AlgQuestions.puskV_questionMVoff.status);

  algoritms_Apusk_status	:= DWORD_TO_UDINT(algoritms.Apusk.status);
  algoritms_Apusk_Start	:= DWORD_TO_UDINT(algoritms.Apusk.Start);
  algoritms_Apusk_Error	:= DWORD_TO_UDINT(algoritms.Apusk.Error);
  algoritms_Apusk_Top	          := DWORD_TO_UDINT(algoritms.Apusk.Top);

  algoritms_SemiAutoPusk_status	:= DWORD_TO_UDINT(algoritms.SemiAutoPusk.status);
  algoritms_SemiAutoPusk_Start	:= DWORD_TO_UDINT(algoritms.SemiAutoPusk.Start);
  algoritms_SemiAutoPusk_Error	:= DWORD_TO_UDINT(algoritms.SemiAutoPusk.Error);
  algoritms_SemiAutoPusk_Top	:= DWORD_TO_UDINT(algoritms.SemiAutoPusk.Top);
  algoritms_SemiAutoPusk_cmdRun1ph_status	:= DWORD_TO_UDINT(AlgQuestions.SemiAutoPusk_cmdRun1ph.status);
  algoritms_SemiAutoPusk_cmdRun2ph_status	:= DWORD_TO_UDINT(AlgQuestions.SemiAutoPusk_cmdRun2ph.status);
  algoritms_SemiAutoPusk_cmdRun3ph_status	:= DWORD_TO_UDINT(AlgQuestions.SemiAutoPusk_cmdRun3ph.status);
  algoritms_SemiAutoPusk_cmdRun4ph_status	:= DWORD_TO_UDINT(AlgQuestions.SemiAutoPusk_cmdRun4ph.status);

  algoritms_AutoPns_status	:= DWORD_TO_UDINT(algoritms.AutoPns.status);
  algoritms_AutoPns_OnTimer	:= AlgTimers.AutoPns_OnTimer;
  algoritms_AutoPns_OffTimer	:= AlgTimers.AutoPns_OffTimer;

  algoritms_autoNu_status	:= DWORD_TO_UDINT(algoritms.autoNu.status);

  algoritms_AutoAvom_status	:= DWORD_TO_UDINT(algoritms.AutoAvom.status);

  algoritms_TestProtection_status	:= DWORD_TO_UDINT(algoritms.TestProtection.status);

  algoritms_Remont_status	:= DWORD_TO_UDINT(algoritms.Remont.status);

  algoritms_AutoTen_status	:= DWORD_TO_UDINT(algoritms.AutoTen.status);
END_FUNCTION_BLOCK

FUNCTION_BLOCK OPC_algoritms_get
  VAR_EXTERNAL
    algoritms : AlgoritmsConfig;
    algoritms_AntiPompag_UgolVNA_inCommand_ARM : UINT;
    algoritms_AntiPompag_zapas_inCommand_ARM : UINT;
    algoritms_Apusk_inCommand_ARM : UINT;
    algoritms_AutoAvom_inCommand_ARM : UINT;
    algoritms_AutoPns_inCommand_ARM : UINT;
    algoritms_AutoTen_inCommand_ARM : UINT;
    algoritms_Remont_inCommand_ARM : UINT;
    algoritms_RingToLine_inCommand_ARM : UINT;
    algoritms_SemiAutoPusk_cmdRun1ph_inCommand_ARM : UINT;
    algoritms_SemiAutoPusk_cmdRun2ph_inCommand_ARM : UINT;
    algoritms_SemiAutoPusk_cmdRun3ph_inCommand_ARM : UINT;
    algoritms_SemiAutoPusk_cmdRun4ph_inCommand_ARM : UINT;
    algoritms_SemiAutoPusk_inCommand_ARM : UINT;
    algoritms_TestProtection_inCommand_ARM : UINT;
    algoritms_ao_inCommand_ARM : UINT;
    algoritms_engineRun_inCommand_ARM : UINT;
    algoritms_filling_inCommand_ARM : UINT;
    algoritms_no_inCommand_ARM : UINT;
    algoritms_ppu_inCommand_ARM : UINT;
    algoritms_puskK_inCommand_ARM : UINT;
    algoritms_puskK_questionFilling_inCommand_ARM : UINT;
    algoritms_puskK_questionUnload_inCommand_ARM : UINT;
    algoritms_puskOilSystem_Ust_dPmg_inCommand_ARM : UINT;
    algoritms_puskOilSystem_inCommand_ARM : UINT;
    algoritms_puskV_inCommand_ARM : UINT;
    algoritms_puskV_questionFilling_inCommand_ARM : UINT;
    algoritms_puskV_questionMVoff_inCommand_ARM : UINT;
    algoritms_testIm_TypeSwitch_inCommand_ARM : UINT;
    algoritms_testIm_inCommand_ARM : UINT;
    algoritms_testPms_algContinue_inCommand_ARM : UINT;
    algoritms_testPms_inCommand_ARM : UINT;
    algoritms_testdPmg_algContinue_inCommand_ARM : UINT;
    algoritms_testdPmg_inCommand_ARM : UINT;
    algoritms_vibegPNS_algContinue_inCommand_ARM : UINT;
    AlgQuestions : AlgoritmsQuestions;
    algoritms_autoNu_inCommand_ARM : UINT;
    algoritms_vibegPNS_inCommand_ARM : UINT;
  END_VAR

  (* OPC Get - algoritms. Чтение текущих состояний тэгов _______________________________________________________*)

  algoritms.ao.inCommand_ARM	:= UINT_TO_WORD(algoritms_ao_inCommand_ARM);

  algoritms.Apusk.inCommand_ARM	:= UINT_TO_WORD(algoritms_Apusk_inCommand_ARM);

  algoritms.AutoAvom.inCommand_ARM	:= UINT_TO_WORD(algoritms_AutoAvom_inCommand_ARM);

  algoritms.autoNu.inCommand_ARM	:= UINT_TO_WORD(algoritms_autoNu_inCommand_ARM);

  algoritms.AutoPns.inCommand_ARM	:= UINT_TO_WORD(algoritms_AutoPns_inCommand_ARM);

  algoritms.engineRun.inCommand_ARM	:= UINT_TO_WORD(algoritms_engineRun_inCommand_ARM);

  algoritms.filling.inCommand_ARM	:= UINT_TO_WORD(algoritms_filling_inCommand_ARM);

  algoritms.no.inCommand_ARM	:= UINT_TO_WORD(algoritms_no_inCommand_ARM);

  algoritms.ppu.inCommand_ARM	:= UINT_TO_WORD(algoritms_ppu_inCommand_ARM);

  AlgQuestions.puskK_questionFilling.inCommand	:= UINT_TO_WORD(algoritms_puskK_questionFilling_inCommand_ARM);
  AlgQuestions.puskK_questionUnload.inCommand	:= UINT_TO_WORD(algoritms_puskK_questionUnload_inCommand_ARM);
  algoritms.puskK.inCommand_ARM	:= UINT_TO_WORD(algoritms_puskK_inCommand_ARM);

  algoritms.puskOilSystem.inCommand_ARM	:= UINT_TO_WORD(algoritms_puskOilSystem_inCommand_ARM);

  AlgQuestions.puskV_questionEngine.inCommand	:= UINT_TO_WORD(algoritms_puskV_questionFilling_inCommand_ARM);
  AlgQuestions.puskV_questionMVoff.inCommand	:= UINT_TO_WORD(algoritms_puskV_questionMVoff_inCommand_ARM);
  algoritms.puskV.inCommand_ARM	:= UINT_TO_WORD(algoritms_puskV_inCommand_ARM);

  algoritms.Remont.inCommand_ARM	:= UINT_TO_WORD(algoritms_Remont_inCommand_ARM);

  algoritms.RingToLine.inCommand_ARM	:= UINT_TO_WORD(algoritms_RingToLine_inCommand_ARM);

  AlgQuestions.SemiAutoPusk_cmdRun1ph.inCommand	:= UINT_TO_WORD(algoritms_SemiAutoPusk_cmdRun1ph_inCommand_ARM);
  AlgQuestions.SemiAutoPusk_cmdRun2ph.inCommand	:= UINT_TO_WORD(algoritms_SemiAutoPusk_cmdRun2ph_inCommand_ARM);
  AlgQuestions.SemiAutoPusk_cmdRun3ph.inCommand	:= UINT_TO_WORD(algoritms_SemiAutoPusk_cmdRun3ph_inCommand_ARM);
  AlgQuestions.SemiAutoPusk_cmdRun4ph.inCommand	:= UINT_TO_WORD(algoritms_SemiAutoPusk_cmdRun4ph_inCommand_ARM);
  algoritms.SemiAutoPusk.inCommand_ARM	:= UINT_TO_WORD(algoritms_SemiAutoPusk_inCommand_ARM);

  AlgQuestions.testdPmg_algContinue.inCommand	:= UINT_TO_WORD(algoritms_testdPmg_algContinue_inCommand_ARM);
  algoritms.testdPmg.inCommand_ARM	:= UINT_TO_WORD(algoritms_testdPmg_inCommand_ARM);

  algoritms.testIm.inCommand_ARM	:= UINT_TO_WORD(algoritms_testIm_inCommand_ARM);

  AlgQuestions.testPms_algContinue.inCommand	:= UINT_TO_WORD(algoritms_testPms_algContinue_inCommand_ARM);
  algoritms.testPms.inCommand_ARM	:= UINT_TO_WORD(algoritms_testPms_inCommand_ARM);

  algoritms.TestProtection.inCommand_ARM	:= UINT_TO_WORD(algoritms_TestProtection_inCommand_ARM);

  AlgQuestions.vibegPNS_algContinue.inCommand	:= UINT_TO_WORD(algoritms_vibegPNS_algContinue_inCommand_ARM);
  algoritms.vibegPNS.inCommand_ARM	:= UINT_TO_WORD(algoritms_vibegPNS_inCommand_ARM);

  algoritms.AutoTen.inCommand_ARM	:= UINT_TO_WORD(algoritms_AutoTen_inCommand_ARM);
END_FUNCTION_BLOCK

FUNCTION_BLOCK fb_Kran_Init
  VAR_INPUT
    data_Ini : BOOL;
    ISVALIDREF_statOn : BOOL;
    ISVALIDREF_statOff : BOOL;
    ISVALIDREF_cmdOn : BOOL;
    ISVALIDREF_cmdOff : BOOL;
    ISVALIDREF_inSo : BOOL;
    ISVALIDREF_inSz : BOOL;
    ISVALIDREF_inDp : BOOL := False;
    continueHoldCommand : TIME;
  END_VAR
  VAR_IN_OUT
    str_Kr : struct_Kran;
  END_VAR
  VAR_OUTPUT
    Init : BOOL := FALSE;
  END_VAR

  (*****            Функциональный блок переинициализации структуры  Kran          *****)

          Init := False;

      IF data_Ini THEN                            (* Параметрам требуется переинициализация. *)
          str_Kr.ISVALIDREF_statOn                := ISVALIDREF_statOn;
          str_Kr.ISVALIDREF_statOff               := ISVALIDREF_statOff;
          str_Kr.ISVALIDREF_cmdOn                 := ISVALIDREF_cmdOn;
          str_Kr.ISVALIDREF_cmdOff                := ISVALIDREF_cmdOff;
          str_Kr.ISVALIDREF_inSo                  := ISVALIDREF_inSo;
          str_Kr.ISVALIDREF_inSz                  := ISVALIDREF_inSz;
          str_Kr.ISVALIDREF_inDp                  := ISVALIDREF_inDp;
          str_Kr.continueHoldCommand              := continueHoldCommand;

          data_Ini:=False;
          Init := TRUE;
     END_IF;
   IF Init THEN
          ISVALIDREF_statOn:= false;
          ISVALIDREF_statOff:= false;
          ISVALIDREF_cmdOn:= false;
          ISVALIDREF_cmdOff:= false;
          ISVALIDREF_inSo:= false;
          ISVALIDREF_inSz:= false;
          ISVALIDREF_inDp:= false;
          continueHoldCommand:= T#0S;
    END_IF;
END_FUNCTION_BLOCK

FUNCTION_BLOCK fb_Switch_Init
  VAR_INPUT
    data_Ini : BOOL;
    ISVALIDREF_statOn : BOOL;
    ISVALIDREF_statOff : BOOL;
    ISVALIDREF_cmdOn : BOOL;
    ISVALIDREF_cmdOff : BOOL;
    ISVALIDREF_inBreakCmdOn : BOOL;
    ISVALIDREF_inBreakCmdOff : BOOL;
  END_VAR
  VAR_IN_OUT
    str_Sw : struct_Switch;
  END_VAR
  VAR_OUTPUT
    Init : BOOL := FALSE;
  END_VAR

  (*****            Функциональный блок переинициализации структуры  Switch          *****)

   Init := FALSE;

      IF data_Ini THEN                            (* Параметрам требуется переинициализация. *)
          str_Sw.ISVALIDREF_statOn                := ISVALIDREF_statOn;
          str_Sw.ISVALIDREF_statOff               := ISVALIDREF_statOff;
          str_Sw.ISVALIDREF_cmdOn                 := ISVALIDREF_cmdOn;
          str_Sw.ISVALIDREF_cmdOff                := ISVALIDREF_cmdOff;
          str_Sw.ISVALIDREF_inBreakCmdOn          := ISVALIDREF_inBreakCmdOn;
          str_Sw.ISVALIDREF_inBreakCmdOff         := ISVALIDREF_inBreakCmdOff;
          data_Ini:=FALSE;
          Init := TRUE;
      END_IF;
  IF Init THEN
          ISVALIDREF_statOn:= FALSE;
          ISVALIDREF_statOff:= FALSE;
          ISVALIDREF_cmdOn:= FALSE;
          ISVALIDREF_cmdOff:= FALSE;
          ISVALIDREF_inBreakCmdOn:= FALSE;
          ISVALIDREF_inBreakCmdOff:= FALSE;
  END_IF;
END_FUNCTION_BLOCK

FUNCTION_BLOCK fb_OilPump_Init
  VAR_INPUT
    data_Ini : BOOL;
    ISVALIDREF_statOn : BOOL;
    ISVALIDREF_statOff : BOOL;
    ISVALIDREF_cmdOn : BOOL;
    ISVALIDREF_cmdOff : BOOL;
    ISVALIDREF_inBreakCmdOn : BOOL;
    ISVALIDREF_inBreakCmdOff : BOOL;
  END_VAR
  VAR_IN_OUT
    str_Op : struct_OilPump;
  END_VAR
  VAR_OUTPUT
    Init : BOOL := FALSE;
  END_VAR

  (*****            Функциональный блок переинициализации структуры  НУ          *****)

   Init := FALSE;

      IF data_Ini THEN                            (* Параметрам требуется переинициализация. *)
          str_Op.ISVALIDREF_statOn                := ISVALIDREF_statOn;
          str_Op.ISVALIDREF_statOff               := ISVALIDREF_statOff;
          str_Op.ISVALIDREF_cmdOn                 := ISVALIDREF_cmdOn;
          str_Op.ISVALIDREF_cmdOff                := ISVALIDREF_cmdOff;
          str_Op.ISVALIDREF_inBreakCmdOn          := ISVALIDREF_inBreakCmdOn;
          str_Op.ISVALIDREF_inBreakCmdOff         := ISVALIDREF_inBreakCmdOff;
          data_Ini:=FALSE;
          Init := TRUE;
      END_IF;

          ISVALIDREF_statOn:= FALSE;
          ISVALIDREF_statOff:= FALSE;
          ISVALIDREF_cmdOn:= FALSE;
          ISVALIDREF_cmdOff:= FALSE;
          ISVALIDREF_inBreakCmdOn:= FALSE;
          ISVALIDREF_inBreakCmdOff:= FALSE;
END_FUNCTION_BLOCK

FUNCTION_BLOCK fb_SectionSwitch_Init
  VAR_INPUT
    data_Ini : BOOL;
    ISVALIDREF_statOn : BOOL;
    ISVALIDREF_statOff : BOOL;
    ISVALIDREF_cmdOn : BOOL;
    ISVALIDREF_cmdOff : BOOL;
    ISVALIDREF_inBreakCmdOn : BOOL;
    ISVALIDREF_inBreakCmdOff : BOOL;
    ISVALIDREF_basketRolledIn : BOOL;
    ISVALIDREF_basketRolledOut : BOOL;
    ISVALIDREF_basketTest : BOOL;
  END_VAR
  VAR_IN_OUT
    str_Sw : struct_SectionSwitch;
  END_VAR
  VAR_OUTPUT
    Init : BOOL := FALSE;
  END_VAR

  (*****            Функциональный блок переинициализации структуры  МВ          *****)

   Init := FALSE;

      IF data_Ini THEN                            (* Параметрам требуется переинициализация. *)
          str_Sw.ISVALIDREF_statOn                := ISVALIDREF_statOn;
          str_Sw.ISVALIDREF_statOff               := ISVALIDREF_statOff;
          str_Sw.ISVALIDREF_cmdOn                 := ISVALIDREF_cmdOn;
          str_Sw.ISVALIDREF_cmdOff                := ISVALIDREF_cmdOff;
          str_Sw.ISVALIDREF_inBreakCmdOn          := ISVALIDREF_inBreakCmdOn;
          str_Sw.ISVALIDREF_inBreakCmdOff         := ISVALIDREF_inBreakCmdOff;
          str_Sw.ISVALIDREF_basketRolledIn        := ISVALIDREF_basketRolledIn;
          str_Sw.ISVALIDREF_basketRolledOut       := ISVALIDREF_basketRolledOut;
          str_Sw.ISVALIDREF_basketTest            := ISVALIDREF_basketTest;
          data_Ini:=FALSE;
          Init := TRUE;
      END_IF;
  IF Init THEN
          ISVALIDREF_statOn:= FALSE;
          ISVALIDREF_statOff:= FALSE;
          ISVALIDREF_cmdOn:= FALSE;
          ISVALIDREF_cmdOff:= FALSE;
          ISVALIDREF_inBreakCmdOn:= FALSE;
          ISVALIDREF_inBreakCmdOff:= FALSE;
          ISVALIDREF_basketRolledIn:= FALSE;
          ISVALIDREF_basketRolledOut:= FALSE;
          ISVALIDREF_basketTest:= FALSE;
  END_IF;
END_FUNCTION_BLOCK

FUNCTION_BLOCK fb_AnalogParametr_Init
  VAR_INPUT
    data_Ini : BOOL;
    currentValue : LREAL;
    minVal : LREAL;
    maxVal : LREAL;
    maxStep : LREAL;
    minVal_ISVALIDREF : BOOL;
    maxVal_ISVALIDREF : BOOL;
    maxStep_ISVALIDREF : BOOL;
  END_VAR
  VAR_IN_OUT
    strAP : struct_AnalogParametr;
  END_VAR
  VAR_OUTPUT
    Init : BOOL := FALSE;
  END_VAR

  (*****            Функциональный блок переинициализации Аналогового параметра.            *****)
       Init := false;

      IF data_Ini THEN                            (* Параметрам требуется переинициализация. *)
          strAP.currentValue          := currentValue;
          strAP.minVal                := minVal;
          strAP.maxVal                := maxVal;
          strAP.maxStep               := maxStep;
          strAP.minVal_ISVALIDREF     := minVal_ISVALIDREF;
          strAP.maxVal_ISVALIDREF     := maxVal_ISVALIDREF;
          strAP.maxStep_ISVALIDREF    := maxStep_ISVALIDREF;

          data_Ini:=false;
          Init := TRUE;
       END_IF;
       IF Init THEN
          currentValue:= 0.0;
          minVal:= 0.0;
          maxVal:= 0.0;
          maxStep:= 0.0;
          minVal_ISVALIDREF:= false;
          maxVal_ISVALIDREF:= false;
          maxStep_ISVALIDREF:= false;
       END_IF;
END_FUNCTION_BLOCK

FUNCTION_BLOCK fb_DiscretParametr_Init
  VAR_INPUT
    data_Ini : BOOL;
    currentValue : UINT;
  END_VAR
  VAR_IN_OUT
    strDp : struct_DiscretParametr;
  END_VAR
  VAR_OUTPUT
    Init : BOOL := FALSE;
  END_VAR

  (*****            Функциональный блок переинициализации дискретного параметра.          *****)

   Init := FALSE;

      IF data_Ini THEN                            (* Параметрам требуется переинициализация. *)
          strDp.currentValue       := currentValue;
          data_Ini:=FALSE;
          Init := TRUE;
      END_IF;
  IF Init THEN
  currentValue:=0;
  END_IF;
END_FUNCTION_BLOCK

FUNCTION_BLOCK fb_singleSignal_Init
  VAR_INPUT
    data_Ini : BOOL;
    inverse : BOOL;
    DelayOn : TIME;
    DelayOff : TIME;
  END_VAR
  VAR_IN_OUT
    str_SS : struct_singleSignal;
  END_VAR
  VAR_OUTPUT
    Init : BOOL := FALSE;
  END_VAR

  (*****            Функциональный блок переинициализации структуры  singleSignal          *****)
  Init := FALSE;

      IF data_Ini THEN                            (* Параметрам требуется переинициализация. *)
          str_SS.inverse                := inverse;
          str_SS.DelayOn                := DelayOn;
          str_SS.DelayOff               := DelayOff;

          data_Ini:=FALSE;
          Init := TRUE;
      END_IF;
   IF Init THEN
          inverse := FALSE;
          DelayOn := T#0S;
          DelayOff:= T#0S;
   END_IF;
END_FUNCTION_BLOCK

FUNCTION_BLOCK fb_singleOutput_Init
  VAR_INPUT
    data_Ini : BOOL;
    inOpcCommandsDisabled : BOOL;
    wait_time : TIME;
  END_VAR
  VAR_IN_OUT
    str_SO : struct_singleOutput;
  END_VAR
  VAR_OUTPUT
    Init : BOOL := FALSE;
  END_VAR

  (*****            Функциональный блок переинициализации структуры  singleOutput          *****)

  Init := FALSE;

      IF data_Ini THEN                            (* Параметрам требуется переинициализация. *)
          str_SO.inOpcCommandsDisabled    := inOpcCommandsDisabled;
          str_SO.wait_time                := wait_time;

           data_Ini:=FALSE;
          Init := TRUE;
      END_IF;
   IF Init THEN
          inOpcCommandsDisabled := FALSE;
          wait_time := T#0S;
     END_IF;
END_FUNCTION_BLOCK

FUNCTION_BLOCK proc_IM_Init
  VAR_INPUT
    init : BOOL;
  END_VAR
  VAR
    stKr_Ini : fb_Kran_Init;
    stSw_Ini : fb_Switch_Init;
    stOp_Ini : fb_OilPump_Init;
    stSSw_Ini : fb_SectionSwitch_Init;
    stAp_Ini : fb_AnalogParametr_Init;
    stDp_Ini : fb_DiscretParametr_Init;
    stSs_Ini : fb_singleSignal_Init;
    stSo_Ini : fb_singleOutput_Init;
    inits : UINT;
  END_VAR
  VAR_INPUT
    initiales : UINT;
  END_VAR
  VAR_EXTERNAL
    IM : ImConfig;
  END_VAR

  inits := 0; (* Флаг необходимости инициализации структур-дескрипторов *)

                                       (* Стартовая инициализация ИМ *)
  (* Кран 1 *)
  stKr_Ini(data_Ini := true, ISVALIDREF_statOn:=true, ISVALIDREF_statOff:=true,
        ISVALIDREF_cmdOn:=true, ISVALIDREF_cmdOff:=true, ISVALIDREF_inDp:=true,
        ISVALIDREF_inSo:=true, ISVALIDREF_inSz:=true,
        str_Kr := IM.Kran1);
  inits := inits + BOOL_TO_UINT(stKr_Ini.Init);

  (* Кран 2 *)
  stKr_Ini(data_Ini := true, ISVALIDREF_statOn:=true, ISVALIDREF_statOff:=true,
        ISVALIDREF_cmdOn:=true, ISVALIDREF_cmdOff:=true,
        ISVALIDREF_inSo:=true, ISVALIDREF_inSz:=true,
        str_Kr := IM.Kran2);
  inits := inits + BOOL_TO_UINT(stKr_Ini.Init);

  (* Кран 3b *)
  stKr_Ini(data_Ini := true, ISVALIDREF_statOn:=true, ISVALIDREF_statOff:=true,
        ISVALIDREF_cmdOn:=true, ISVALIDREF_cmdOff:=true,
        ISVALIDREF_inSo:=true, ISVALIDREF_inSz:=true, continueHoldCommand:=T#5S,
        str_Kr := IM.Kran3b);
  inits := inits + BOOL_TO_UINT(stKr_Ini.Init);

  (* Кран 4 *)
  stKr_Ini(data_Ini := true, ISVALIDREF_statOn:=true, ISVALIDREF_statOff:=true,
        ISVALIDREF_cmdOn:=true, ISVALIDREF_cmdOff:=true,
        ISVALIDREF_inSo:=true, ISVALIDREF_inSz:=true,
        str_Kr := IM.Kran4);
  inits := inits + BOOL_TO_UINT(stKr_Ini.Init);

  (* Кран 5 *)
  stKr_Ini(data_Ini := true, ISVALIDREF_statOn:=true, ISVALIDREF_statOff:=true,
        ISVALIDREF_cmdOn:=true, ISVALIDREF_cmdOff:=true,
        ISVALIDREF_inSo:=true, ISVALIDREF_inSz:=true, continueHoldCommand:=T#5S,
        str_Kr := IM.Kran5);
  inits := inits + BOOL_TO_UINT(stKr_Ini.Init);

  (* Кран 6 *)
  stKr_Ini(data_Ini := true, ISVALIDREF_statOn:=true, ISVALIDREF_statOff:=true,
        ISVALIDREF_cmdOn:=true, ISVALIDREF_cmdOff:=true,
        str_Kr := IM.Kran6);
  inits := inits + BOOL_TO_UINT(stKr_Ini.Init);

  (* НУ1 Насос уплотнения *)
  stOp_Ini(data_Ini := true, ISVALIDREF_statOn:=true, (*ISVALIDREF_statOff:=true,*)
        ISVALIDREF_cmdOn:=true, ISVALIDREF_cmdOff:=true,
        ISVALIDREF_inBreakCmdOn:=true, (*ISVALIDREF_inBreakCmdOff:=true,*)
        str_Op := IM.nu1);
  inits := inits + BOOL_TO_UINT(stOp_Ini.Init);

  (* НУ2 Насос уплотнения *)
  stOp_Ini(data_Ini := true, ISVALIDREF_statOn:=true, (*ISVALIDREF_statOff:=true,*)
        ISVALIDREF_cmdOn:=true, ISVALIDREF_cmdOff:=true,
        ISVALIDREF_inBreakCmdOn:=true, (*ISVALIDREF_inBreakCmdOff:=true,*)
        str_Op := IM.nu2);
  inits := inits + BOOL_TO_UINT(stOp_Ini.Init);

  (* ПНС Насос смазки *)
  stSw_Ini(data_Ini := true, ISVALIDREF_statOn:=true, (*ISVALIDREF_statOff:=true,*)
        ISVALIDREF_cmdOn:=true, ISVALIDREF_cmdOff:=true,
        ISVALIDREF_inBreakCmdOn:=true, (*ISVALIDREF_inBreakCmdOff:=true,*)
        str_Sw := IM.pns);
  inits := inits + BOOL_TO_UINT(stSw_Ini.Init);

  (* В1 АВОМ вентилятор охлаждения *)
  stSw_Ini(data_Ini := true, ISVALIDREF_statOn:=true, (*ISVALIDREF_statOff:=true,*)
        ISVALIDREF_cmdOn:=true, ISVALIDREF_cmdOff:=true,
        ISVALIDREF_inBreakCmdOn:=true, (*ISVALIDREF_inBreakCmdOff:=true,*)
        str_Sw := IM.v1_Avom);
  inits := inits + BOOL_TO_UINT(stSw_Ini.Init);

  (* В2 АВОМ вентилятор охлаждения *)
  stSw_Ini(data_Ini := true, ISVALIDREF_statOn:=true, (*ISVALIDREF_statOff:=true,*)
        ISVALIDREF_cmdOn:=true, ISVALIDREF_cmdOff:=true,
        ISVALIDREF_inBreakCmdOn:=true, (*ISVALIDREF_inBreakCmdOff:=true,*)
        str_Sw := IM.v2_Avom);
  inits := inits + BOOL_TO_UINT(stSw_Ini.Init);

  (* ТЭН *)
  stSw_Ini(data_Ini := true, ISVALIDREF_statOn:=true, ISVALIDREF_statOff:=true,
        ISVALIDREF_cmdOn:=true, ISVALIDREF_cmdOff:=true,
        (*ISVALIDREF_inBreakCmdOn:=true, ISVALIDREF_inBreakCmdOff:=true,*)
        str_Sw := IM.Ten);
  inits := inits + BOOL_TO_UINT(stSw_Ini.Init);

  (* МВ масляный выключатель *)
  stSSw_Ini(data_Ini := true, (*ISVALIDREF_statOn:=true,*) ISVALIDREF_statOff:=true,
        ISVALIDREF_cmdOn:=true, ISVALIDREF_cmdOff:=true,
        (*ISVALIDREF_inBreakCmdOn:=true,*) ISVALIDREF_inBreakCmdOff:=true,
        ISVALIDREF_basketRolledIn:=true, ISVALIDREF_basketRolledout:=true,
        str_Sw := IM.mv);
  inits := inits + BOOL_TO_UINT(stSSw_Ini.Init);

                                       (* Стартовая инициализация Аналоговых и Дискретных параметров *)

  (* Температура включения АВОМ1 в алгоритме АвтоАвом *)
  stAp_Ini(data_Ini := true, currentValue:=40.0,
        minVal_ISVALIDREF:=true, maxVal_ISVALIDREF:=true,
        minVal:=-50.0, maxVal:=150.0,
        strAP := IM.AutoAvom_onTemp1);
  inits := inits + BOOL_TO_UINT(stAp_Ini.Init);

  (* Температура включения АВОМ2 в алгоритме АвтоАвом *)
  stAp_Ini(data_Ini := true, currentValue:=50.0,
        minVal_ISVALIDREF:=true, maxVal_ISVALIDREF:=true,
        minVal:=-50.0, maxVal:=150.0,
        strAP := IM.AutoAvom_onTemp2);
  inits := inits + BOOL_TO_UINT(stAp_Ini.Init);

  (* Гистерезис уставок теммпературы в алгоритме АвтоАвом *)
  stAp_Ini(data_Ini := true, currentValue:=2.0,
        minVal_ISVALIDREF:=true, maxVal_ISVALIDREF:=true,
        minVal:=0.0, maxVal:=100.0,
        strAP := IM.AutoAvom_hysteresis);
   inits := inits + BOOL_TO_UINT(stAp_Ini.Init);

  (* Давление включения ПНС в алгоритме АвтоПНС *)
  stAp_Ini(data_Ini := true, currentValue:=40.0,
        minVal_ISVALIDREF:=true, maxVal_ISVALIDREF:=true,
        minVal:=0.0, maxVal:=400.0,
        strAP := IM.AutoPns_UstRun);
  inits := inits + BOOL_TO_UINT(stAp_Ini.Init);

  (* Давление отключения ПНС в алгоритме АвтоПНС *)
  stAp_Ini(data_Ini := true, currentValue:=80.0,
        minVal_ISVALIDREF:=true, maxVal_ISVALIDREF:=true,
        minVal:=0.0, maxVal:=400.0,
        strAP := IM.AutoPns_UstStop);
   inits := inits + BOOL_TO_UINT(stAp_Ini.Init);

  (* Давление масло-газ включения защит в алгоритме Пуск Маслосистемы *)
  stAp_Ini(data_Ini := true, currentValue:=100.0,
        minVal_ISVALIDREF:=true, maxVal_ISVALIDREF:=true,
        minVal:=0.0, maxVal:=630.0,
        strAP := IM.PuskOilSystem_UstdPmg);
   inits := inits + BOOL_TO_UINT(stAp_Ini.Init);

   (* Температура отключения ТЭНа в алгоритме АвтоТЭН *)
  stAp_Ini(data_Ini := true, currentValue:=20.0,
        minVal_ISVALIDREF:=true, maxVal_ISVALIDREF:=true,
        minVal:=-50.0, maxVal:=150.0,
        strAP := IM.AutoTen_offTemperature);
   inits := inits + BOOL_TO_UINT(stAp_Ini.Init);

    (* Уставка включения резервного НУ по перепаду давления "масло-газ" в алгоритме АвтоНУ *)
  stAp_Ini(data_Ini := true, currentValue:=105.0,
        minVal_ISVALIDREF:=true, maxVal_ISVALIDREF:=true,
        minVal:=0.0, maxVal:=630.0,
        strAP := IM.AutoNU_Ust_Swap);
   inits := inits + BOOL_TO_UINT(stAp_Ini.Init);

   (* Уставка по перепаду давления "масло-газ" в алгоритме Тест dPmg *)
  stAp_Ini(data_Ini := true, currentValue:=100.0,
        minVal_ISVALIDREF:=true, maxVal_ISVALIDREF:=true,
        minVal:=0.0, maxVal:=630.0,
        strAP := IM.testdPmg_Ust_dPLow);
   inits := inits + BOOL_TO_UINT(stAp_Ini.Init);

    (* Угол наклона ВНА в алгоритме Антипомпаж *)
  stAp_Ini(data_Ini := true, currentValue:=0.0,
        minVal_ISVALIDREF:=true, maxVal_ISVALIDREF:=true,
        minVal:=-35.0, maxVal:=35.0,
        strAP := IM.AntiPompag_UgolVNA);
   inits := inits + BOOL_TO_UINT(stAp_Ini.Init);

    (*Коэффициент сжимаемости газа в алгоритме Антипомпаж *)
  stAp_Ini(data_Ini := true, currentValue:=0.94,
        strAP := IM.AntiPompag_K);
   inits := inits + BOOL_TO_UINT(stAp_Ini.Init);

    (*Коэффициент расхода конфузора в алгоритме Антипомпаж *)
  stAp_Ini(data_Ini := true, currentValue:=68.4,
        strAP := IM.AntiPompag_A);
   inits := inits + BOOL_TO_UINT(stAp_Ini.Init);

    (*Удельный вес газа в алгоритме Антипомпаж *)
  stAp_Ini(data_Ini := true, currentValue:=0.73,
        strAP := IM.AntiPompag_y0);
   inits := inits + BOOL_TO_UINT(stAp_Ini.Init);

  (* Переключатель разблокировки кранов: 1 - допстить управление кранами *)
  stDp_Ini(data_Ini := true, currentValue:=0,
        strDp := IM.TypeSwitch);
  inits := inits + BOOL_TO_UINT(stDp_Ini.Init);

  (* Селектор выбора основной/резервный НУ *)
  stDp_Ini(data_Ini := true, currentValue:=0,
        strDp := IM.AutoNU_mainNU);
  inits := inits + BOOL_TO_UINT(stDp_Ini.Init);

                                       (* Стартовая инициализация singleSignal *)

      (* Перепад давления «газ-газ» на кране 1 ≤1 кгс/см² *)
  stSs_Ini(data_Ini := true, inverse:=FALSE, (*DelayOn:=T#0S, DelayOff:=T#0S,*) str_SS := IM.SingleSignals.dP_gazgaz_Kran1);
  inits := inits + BOOL_TO_UINT(stSs_Ini.Init);

   (* Осевой сдвиг ротора вправо ≥3,7 кгс/см² *)
  stSs_Ini(data_Ini := true, inverse:=FALSE, (*DelayOn:=T#0S, DelayOff:=T#0S,*) str_SS := IM.SingleSignals.OsevoiSdvig_pravo);
  inits := inits + BOOL_TO_UINT(stSs_Ini.Init);

   (* Осевой сдвиг ротора влево ≥3,7 кгс/см² *)
  stSs_Ini(data_Ini := true, inverse:=FALSE, (*DelayOn:=T#0S, DelayOff:=T#0S,*) str_SS := IM.SingleSignals.OsevoiSdvig_levo);
  inits := inits + BOOL_TO_UINT(stSs_Ini.Init);

   (* Низкий перепад давления «масло-газ» ≤1 кгс/см² *)
  stSs_Ini(data_Ini := true, inverse:=FALSE, (*DelayOn:=T#0S, DelayOff:=T#0S,*) str_SS := IM.SingleSignals.dP_oilgaz_low);
  inits := inits + BOOL_TO_UINT(stSs_Ini.Init);

  (* Низкое давление масла смазки ≤ 0,4 кгс/см² *)
  stSs_Ini(data_Ini := true, inverse:=FALSE, (*DelayOn:=T#0S, DelayOff:=T#0S,*) str_SS := IM.SingleSignals.P_oil_low);
  inits := inits + BOOL_TO_UINT(stSs_Ini.Init);

      (* Защита по замыканию на землю 10 кВ (пробой изоляции кабелей) *)
  stSs_Ini(data_Ini := true, inverse:=FALSE, (*DelayOn:=T#0S, DelayOff:=T#0S,*) str_SS := IM.SingleSignals.KZ_10kv);
  inits := inits + BOOL_TO_UINT(stSs_Ini.Init);

      (* Пробой вентиля *)
  stSs_Ini(data_Ini := true, inverse:=TRUE, (*DelayOn:=T#0S, DelayOff:=T#0S,*) str_SS := IM.SingleSignals.Vozb_ProboiVentila);
  inits := inits + BOOL_TO_UINT(stSs_Ini.Init);

      (* Асинхронный ход и перегрузка *)
  stSs_Ini(data_Ini := true, inverse:=TRUE, (*DelayOn:=T#0S, DelayOff:=T#0S,*) str_SS := IM.SingleSignals.Vozb_AsinchHod);
  inits := inits + BOOL_TO_UINT(stSs_Ini.Init);

      (* Работа схемы ресинхронизации *)
  stSs_Ini(data_Ini := true, inverse:=FALSE, (*DelayOn:=T#0S, DelayOff:=T#0S,*) str_SS := IM.SingleSignals.Vozb_ReSynchronize);
  inits := inits + BOOL_TO_UINT(stSs_Ini.Init);

      (* Контроль состояния возбудительного устройства  *)
  stSs_Ini(data_Ini := true, inverse:=FALSE, (*DelayOn:=T#0S, DelayOff:=T#0S,*) str_SS := IM.SingleSignals.Vozb_ControlVozbuditela);
  inits := inits + BOOL_TO_UINT(stSs_Ini.Init);

      (* Неисправность форсировки воз-буждения  *)
  stSs_Ini(data_Ini := true, inverse:=FALSE, (*DelayOn:=T#0S, DelayOff:=T#0S,*) str_SS := IM.SingleSignals.NS_ForsingVozbugdenia);
  inits := inits + BOOL_TO_UINT(stSs_Ini.Init);

    (* Неисправность возбудительного устройства  *)
  stSs_Ini(data_Ini := true, inverse:=FALSE, (*DelayOn:=T#0S, DelayOff:=T#0S,*) str_SS := IM.SingleSignals.NS_Vozbyditela);
  inits := inits + BOOL_TO_UINT(stSs_Ini.Init);

    (* Отключен АВР  *)
  stSs_Ini(data_Ini := true, inverse:=FALSE, (*DelayOn:=T#0S, DelayOff:=T#0S,*) str_SS := IM.SingleSignals.Vozb_AVR_off);
  inits := inits + BOOL_TO_UINT(stSs_Ini.Init);

    (* Отключено автоматическое управление возбудителем  *)
  stSs_Ini(data_Ini := true, inverse:=FALSE, (*DelayOn:=T#0S, DelayOff:=T#0S,*) str_SS := IM.SingleSignals.Vozb_AutoUprVozbuditela_off);
  inits := inits + BOOL_TO_UINT(stSs_Ini.Init);

    (* Контактор возбуждения включен  *)
  stSs_Ini(data_Ini := true, inverse:=TRUE, (*DelayOn:=T#0S, DelayOff:=T#0S,*) str_SS := IM.SingleSignals.Vozb_KontaktorON);
  inits := inits + BOOL_TO_UINT(stSs_Ini.Init);

    (* Перегрузка  *)
  stSs_Ini(data_Ini := true, inverse:=FALSE, (*DelayOn:=T#0S, DelayOff:=T#0S,*) str_SS := IM.SingleSignals.Vozb_Overload);
  inits := inits + BOOL_TO_UINT(stSs_Ini.Init);

    (* Аварийный останов цеха  *)
  stSs_Ini(data_Ini := true, inverse:=FALSE, (*DelayOn:=T#0S, DelayOff:=T#0S,*) str_SS := IM.SingleSignals.AO_KC);
  inits := inits + BOOL_TO_UINT(stSs_Ini.Init);

    (* АО ГПА от кнопки на ПРУ  *)
  stSs_Ini(data_Ini := true, inverse:=FALSE, (*DelayOn:=T#0S, DelayOff:=T#0S,*) str_SS := IM.SingleSignals.AOGPA_PRU);
  inits := inits + BOOL_TO_UINT(stSs_Ini.Init);

    (* Готовность включения БЭО по отказу контроллера  *)
  stSs_Ini(data_Ini := true, inverse:=FALSE, (*DelayOn:=T#0S, DelayOff:=T#0S,*) str_SS := IM.SingleSignals.BEO_Ready);
  inits := inits + BOOL_TO_UINT(stSs_Ini.Init);

    (* Срабатывание БЭАО  *)
  stSs_Ini(data_Ini := true, inverse:=FALSE, (*DelayOn:=T#0S, DelayOff:=T#0S,*) str_SS := IM.SingleSignals.BEO_Srabat);
  inits := inits + BOOL_TO_UINT(stSs_Ini.Init);

    (* Запуск БЭАО от кнопки ЭАО ШУ  *)
  stSs_Ini(data_Ini := true, inverse:=FALSE, (*DelayOn:=T#0S, DelayOff:=T#0S,*) str_SS := IM.SingleSignals.BEO_ON_knopkaSHU);
  inits := inits + BOOL_TO_UINT(stSs_Ini.Init);

    (* Экстренный аварийный останов ЭАО ЭГПА с ПРУ   *)
  stSs_Ini(data_Ini := true, inverse:=FALSE, (*DelayOn:=T#0S, DelayOff:=T#0S,*) str_SS := IM.SingleSignals.BEO_ON_knopkaPRU);
  inits := inits + BOOL_TO_UINT(stSs_Ini.Init);

    (* НО ГПА от ШУ   *)
  stSs_Ini(data_Ini := true, inverse:=FALSE, (*DelayOn:=T#0S, DelayOff:=T#0S,*) str_SS := IM.SingleSignals.NOGPA_knopkaSHU);
  inits := inits + BOOL_TO_UINT(stSs_Ini.Init);

    (* АО ГПА от ШУ   *)
  stSs_Ini(data_Ini := true, inverse:=FALSE, (*DelayOn:=T#0S, DelayOff:=T#0S,*) str_SS := IM.SingleSignals.AOGPA_knopkaSHU);
  inits := inits + BOOL_TO_UINT(stSs_Ini.Init);

    (* Дверь шкафа открыта   *)
  stSs_Ini(data_Ini := true, inverse:=TRUE, (*DelayOn:=T#0S, DelayOff:=T#0S,*) str_SS := IM.SingleSignals.DverShkafaOtkryta);
  inits := inits + BOOL_TO_UINT(stSs_Ini.Init);

    (* Выключатель основного ввода питания QF1  в положении включен   *)
  stSs_Ini(data_Ini := true, inverse:=TRUE, (*DelayOn:=T#0S, DelayOff:=T#0S,*) str_SS := IM.SingleSignals.QF1_on);
  inits := inits + BOOL_TO_UINT(stSs_Ini.Init);

    (* Выключатель резервного ввода питания QF2  в положении включен   *)
  stSs_Ini(data_Ini := true, inverse:=TRUE, (*DelayOn:=T#0S, DelayOff:=T#0S,*) str_SS := IM.SingleSignals.QF2_on);
  inits := inits + BOOL_TO_UINT(stSs_Ini.Init);

    (* Выключатель питания кранов:  QF23 110 В в положении включен   *)
  stSs_Ini(data_Ini := true, inverse:=TRUE, (*DelayOn:=T#0S, DelayOff:=T#0S,*) str_SS := IM.SingleSignals.QF23_on);
  inits := inits + BOOL_TO_UINT(stSs_Ini.Init);

    (* Выключатели группы 1: QF4, QF5 в положении включен   *)
  stSs_Ini(data_Ini := true, inverse:=TRUE, (*DelayOn:=T#0S, DelayOff:=T#0S,*) str_SS := IM.SingleSignals.QF4_QF5_on);
  inits := inits + BOOL_TO_UINT(stSs_Ini.Init);

    (* Выключатели группы 2: QF6, QF7 в положении включен   *)
  stSs_Ini(data_Ini := true, inverse:=TRUE, (*DelayOn:=T#0S, DelayOff:=T#0S,*) str_SS := IM.SingleSignals.QF6_QF7_on);
  inits := inits + BOOL_TO_UINT(stSs_Ini.Init);

    (* Выключатели группы 3: QF8, QF9 в положении включен   *)
  stSs_Ini(data_Ini := true, inverse:=TRUE, (*DelayOn:=T#0S, DelayOff:=T#0S,*) str_SS := IM.SingleSignals.QF8_QF9_on);
  inits := inits + BOOL_TO_UINT(stSs_Ini.Init);

    (* Выключатели группы 4: QF10, QF11 в положении включен   *)
  stSs_Ini(data_Ini := true, inverse:=TRUE, (*DelayOn:=T#0S, DelayOff:=T#0S,*) str_SS := IM.SingleSignals.QF10_QF11_on);
  inits := inits + BOOL_TO_UINT(stSs_Ini.Init);

    (* Выключатели группы 5: QF12, QF13 в положении включен   *)
  stSs_Ini(data_Ini := true, inverse:=TRUE, (*DelayOn:=T#0S, DelayOff:=T#0S,*) str_SS := IM.SingleSignals.QF12_QF13_on);
  inits := inits + BOOL_TO_UINT(stSs_Ini.Init);

    (* Выключатели группы 6: QF14, QF15 в положении включен   *)
  stSs_Ini(data_Ini := true, inverse:=TRUE, (*DelayOn:=T#0S, DelayOff:=T#0S,*) str_SS := IM.SingleSignals.QF14_QF15_on);
  inits := inits + BOOL_TO_UINT(stSs_Ini.Init);

    (* Выключатели группы : QF22 в положении включен   *)
  stSs_Ini(data_Ini := true, inverse:=TRUE, (*DelayOn:=T#0S, DelayOff:=T#0S,*) str_SS := IM.SingleSignals.QF22_on);
  inits := inits + BOOL_TO_UINT(stSs_Ini.Init);

    (* Неисправность источников питания группы 1: G1, G2 (=24 В)   *)
  stSs_Ini(data_Ini := true, inverse:=TRUE, (*DelayOn:=T#0S, DelayOff:=T#0S,*) str_SS := IM.SingleSignals.NS_G1_G2);
  inits := inits + BOOL_TO_UINT(stSs_Ini.Init);

    (* Неисправность источников питания группы 2: G3, G4 (=24 В)   *)
  stSs_Ini(data_Ini := true, inverse:=TRUE, (*DelayOn:=T#0S, DelayOff:=T#0S,*) str_SS := IM.SingleSignals.NS_G3_G4);
  inits := inits + BOOL_TO_UINT(stSs_Ini.Init);

    (* Неисправность источников питания внутренних ПТС: G15, G16 (=24 В)   *)
  stSs_Ini(data_Ini := true, inverse:=TRUE, (*DelayOn:=T#0S, DelayOff:=T#0S,*) str_SS := IM.SingleSignals.NS_G15_G16);
  inits := inits + BOOL_TO_UINT(stSs_Ini.Init);

    (* Неисправность источника питания аналоговых сигналов: G17 (=24 В)   *)
  stSs_Ini(data_Ini := true, inverse:=TRUE, (*DelayOn:=T#0S, DelayOff:=T#0S,*) str_SS := IM.SingleSignals.NS_G17);
  inits := inits + BOOL_TO_UINT(stSs_Ini.Init);

    (* Неисправность источников питания группы 3: G5, G6 (=24 В)   *)
  stSs_Ini(data_Ini := true, inverse:=TRUE, (*DelayOn:=T#0S, DelayOff:=T#0S,*) str_SS := IM.SingleSignals.NS_G5_G6);
  inits := inits + BOOL_TO_UINT(stSs_Ini.Init);

    (* Неисправность источников питания группы 4: G7, G8 (=24 В)   *)
  stSs_Ini(data_Ini := true, inverse:=TRUE, (*DelayOn:=T#0S, DelayOff:=T#0S,*) str_SS := IM.SingleSignals.NS_G7_G8);
  inits := inits + BOOL_TO_UINT(stSs_Ini.Init);

    (* Неисправность источников питания внешних цепей: G18, G19 (=24 В)   *)
  stSs_Ini(data_Ini := true, inverse:=TRUE, (*DelayOn:=T#0S, DelayOff:=T#0S,*) str_SS := IM.SingleSignals.NS_G18_G19);
  inits := inits + BOOL_TO_UINT(stSs_Ini.Init);

    (* Неисправность источников питания группы 5: G9, G10, G11, G12 (=110 В)   *)
  stSs_Ini(data_Ini := true, inverse:=TRUE, (*DelayOn:=T#0S, DelayOff:=T#0S,*) str_SS := IM.SingleSignals.NS_G10_G11);
  inits := inits + BOOL_TO_UINT(stSs_Ini.Init);

    (* Неисправность источников питания G13, G14 (=24 В)   *)
  stSs_Ini(data_Ini := true, inverse:=TRUE, (*DelayOn:=T#0S, DelayOff:=T#0S,*) str_SS := IM.SingleSignals.NS_G13_G14);
  inits := inits + BOOL_TO_UINT(stSs_Ini.Init);

                                       (* Стартовая инициализация singleOutput *)

  (* Идикация НО (подсветка кнопки на шкафу)   *)
  stSo_Ini(data_Ini := true, inOpcCommandsDisabled:=TRUE, (*wait_time:=T#0S,*) str_SO := IM.SingleOutputs.Lampa_NO);
  inits := inits + BOOL_TO_UINT(stSo_Ini.Init);

  (* Взвод включения БЭАО по неисправности ПТС   *)
  stSo_Ini(data_Ini := true, inOpcCommandsDisabled:=TRUE, wait_time:=T#2S, str_SO := IM.SingleOutputs.VzvodBREO);
  inits := inits + BOOL_TO_UINT(stSo_Ini.Init);

  (* Авария ЭГПА в КЦ   *)
  stSo_Ini(data_Ini := true, inOpcCommandsDisabled:=TRUE, (*wait_time:=T#0S,*) str_SO := IM.SingleOutputs.AO_GPA);
  inits := inits + BOOL_TO_UINT(stSo_Ini.Init);

  (* Сброс включения БЭАО по неисправности ПТС   *)
  stSo_Ini(data_Ini := true, inOpcCommandsDisabled:=TRUE, wait_time:=T#2S, str_SO := IM.SingleOutputs.SbrosBREO);
  inits := inits + BOOL_TO_UINT(stSo_Ini.Init);

  (* Индикация ПС Фонарь   *)
  stSo_Ini(data_Ini := true, inOpcCommandsDisabled:=TRUE, (*wait_time:=T#0S,*) str_SO := IM.SingleOutputs.IndikicijaPS_fonar);
  inits := inits + BOOL_TO_UINT(stSo_Ini.Init);

  (* Индикация АС Фонарь   *)
  stSo_Ini(data_Ini := true, inOpcCommandsDisabled:=TRUE, (*wait_time:=T#0S,*) str_SO := IM.SingleOutputs.IndikicijaAS_fonar);
  inits := inits + BOOL_TO_UINT(stSo_Ini.Init);

  (* Отключение МВ1 от КНА   *)
  stSo_Ini(data_Ini := true, inOpcCommandsDisabled:=TRUE, (*wait_time:=T#0S,*) str_SO := IM.SingleOutputs.mv_off_KNA);
  inits := inits + BOOL_TO_UINT(stSo_Ini.Init);

  initiales := 0;
  IF init THEN initiales := inits; END_IF;
END_FUNCTION_BLOCK

FUNCTION_BLOCK fb_Kran
  VAR_INPUT
    statOn : BOOL;
    statOff : BOOL;
    statOn_reliability : BOOL;
    statOff_reliability : BOOL;
  END_VAR
  VAR_IN_OUT
    strKr : struct_Kran;
  END_VAR
  VAR_INPUT
    inNs : TYPE_ReliableBit;
    inAccident : TYPE_ReliableBit;
    inAuto : TYPE_ReliableBit;
    inManual : TYPE_ReliableBit;
    inLocal : TYPE_ReliableBit;
    inDistance : TYPE_ReliableBit;
    inErrorPowerOff : TYPE_ReliableBit;
    inErrorBlock : TYPE_ReliableBit;
    inSo : TYPE_ReliableBit;
    inSz : TYPE_ReliableBit;
    inDp : TYPE_ReliableBit;
  END_VAR
  VAR
    onInit : BOOL := FALSE;
    _statOn : BOOL;
    _statOff : BOOL;
    getSdvig : BOOL;
    lastOnStatus : BYTE;
    cmd : BYTE;
    source : BYTE;
    lastCmd : BYTE;
    source_for_Status : BYTE;
    cmd_for_Status : BYTE;
    command_error_for_Status : BYTE;
    _sunpackerCommand : fb_sunpackerCommand;
    _statusDualInput : TYPE_statusDualInput;
    _commandDualInput : TYPE_commandDualInput;
    _commandErrorTimer : BOOL;
    resetErrorTimer : BOOL;
    _changWithoutCommand : BOOL;
    BlockedOpenControl : BOOL;
    errorCMDTimer : TON;
    _errorReset : TON;
    sdvigReset : TON;
    continueHoldCommandTimer : TON;
    outputsSets : TOF;
    dP_Trig : R_TRIG;
    dP_Trig_reliability : R_TRIG;
    resetBlockedOpenControl_Trig : R_TRIG;
  END_VAR
  VAR_IN_OUT
    cmdOn : BOOL;
    cmdOff : BOOL;
  END_VAR

  IF NOT onInit THEN
  IF strKr.ISVALIDREF_cmdOn XOR strKr.ISVALIDREF_cmdOff THEN
  	IF 	strKr.ISVALIDREF_cmdOn THEN
  		lastCmd:= 2; (*baseCmdOff*)
  	ELSE
  		lastCmd:= 1; (*baseCmdOn*)
  	END_IF;
  END_IF;
  onInit:=TRUE;
  END_IF;

  (* ---- Если управление с ВУ заблокировано, то в ИМ передаем команду из алгоритма ---- *)
  IF strKr.inOpcCommandsDisabled THEN
  	strKr.inCommand := strKr.inCommand_Alg;
  ELSE (* иначе передаем команду с АРМа*)
  	strKr.inCommand := strKr.inCommand_ARM;
  END_IF;

  (* ---- Формирование состояния механизма ---- *)

  IF (strKr.ISVALIDREF_statOn) OR (strKr.ISVALIDREF_statOff) THEN
  	IF (strKr.ISVALIDREF_statOn) AND (strKr.ISVALIDREF_statOff) THEN
  	strKr.reliability:= statOn_reliability AND statOff_reliability;
  		_statOn  := statOn;
  		_statOff := statOff;
  	ELSIF (strKr.ISVALIDREF_statOn) THEN
                       strKr.reliability:= statOn_reliability;
  		_statOn  := statOn;
  		_statOff := NOT statOn;
  	ELSIF (strKr.ISVALIDREF_statOff) THEN
  		 strKr.reliability:= statOff_reliability;
  		_statOn  := NOT statOff;
  		_statOff :=statOff;
  	END_IF;

  	IF strKr.reliability THEN
  		IF _statOn AND NOT _statOff 		THEN 	strKr.onStatus := _statusDualInput.STATUS_ON;
  		ELSIF _statOff AND NOT _statOn 	THEN 	strKr.onStatus := _statusDualInput.Status_OFF;
  		ELSIF NOT _statOn AND NOT _statOff 	THEN 	strKr.onStatus := _statusDualInput.STATUS_TRANSITIONAL;
  		ELSE					strKr.onStatus := _statusDualInput.STATUS_ERROR;
                      END_IF;

  	ELSE
  		strKr.onStatus := _statusDualInput.STATUS_NOTDEFINED;

  	END_IF;
  ELSE
  	CASE BYTE_TO_INT(lastCmd) OF
  		(*baseCmdOn*)  1: strKr.onStatus  := _statusDualInput.STATUS_ON;
  		(*baseCmdOff*) 2: strKr.onStatus  := _statusDualInput.STATUS_OFF;

  	ELSE
  		 strKr.onStatus := _statusDualInput.STATUS_NOTDEFINED;

  	END_CASE;
  END_IF;

  strKr.Accident := inAccident.value AND inAccident.reliability;
  strKr.Ns := inNs.value AND inNs.reliability;
  strKr.Auto := inAuto.value AND inAuto.reliability;
  strKr.Manual := inManual.value AND inManual.reliability;
  strKr.Local := inLocal.value AND inLocal.reliability;
  strKr.Distance := inDistance.value AND inDistance.reliability;
  strKr.ErrorPowerOff := inErrorPowerOff.value AND inErrorPowerOff.reliability;
  strKr.ErrorBlock := inErrorBlock.value AND inErrorBlock.reliability;
  strKr.OpcCommandsDisabled := strKr.inOpcCommandsDisabled;

  (* ---- Формирование признака блокировки Открытия крана по высокому давлению ---- *)
  	IF strKr.ISVALIDREF_inDp THEN

  		strKr.Dp := NOT inDp.value AND inDp.reliability;

  		dP_Trig(CLK := strKr.Dp );
  		dP_Trig_reliability(CLK :=NOT inDp.reliability);

  		IF dP_Trig.Q OR dP_Trig_reliability.Q THEN
  			BlockedOpenControl := TRUE;
  		END_IF;
  		(* ---- автоматический сброс *)
  		resetBlockedOpenControl_Trig(CLK := (inDp.value) AND inDp.reliability);
  		IF resetBlockedOpenControl_Trig.Q THEN
  			BlockedOpenControl := FALSE;
  		END_IF;
  	ELSE
  		strKr.Dp  := FALSE;
  		BlockedOpenControl := FALSE;
  	END_IF;

  (* ---- Формирование признака сдвига ---- *)
  getSdvig := FALSE;
  IF (strKr.ISVALIDREF_cmdOn OR strKr.ISVALIDREF_cmdOff) AND NOT strKr.Local THEN
  	IF NOT (strKr.CmdOn OR strKr.CmdOff) THEN
  		IF (lastOnStatus <> strKr.onStatus AND
  		(strKr.onStatus <> _statusDualInput.STATUS_NOTDEFINED AND strKr.onStatus <> _statusDualInput.STATUS_ERROR) AND
  		(lastOnStatus <> _statusDualInput.STATUS_NOTDEFINED AND lastOnStatus <> _statusDualInput.STATUS_ERROR)) THEN
  			strKr.sdvig   := TRUE;
  		END_IF;
  	END_IF;
  END_IF;

  IF getSdvig THEN strKr.sdvig:= TRUE; END_IF;

  sdvigReset(IN:=strKr.sdvig, PT:=T#15S);

  IF sdvigReset.Q THEN strKr.sdvig:=FALSE; END_IF;

  lastOnStatus := strKr.onStatus;

  (* ---- Распаковка команды ---- *)
  _sunpackerCommand(command := strKr.inCommand);
  	cmd := _sunpackerCommand.cmd;
  	source := _sunpackerCommand.source;

  (* ---- Обработка команды ---- *)
  IF cmd <> 0 AND lastCmd <> cmd and (((NOT strKr.opcCommandsDisabled) AND source > 0) OR source = 0) then
  	CASE BYTE_TO_INT(cmd) OF
  	(*cmd_open*) 1 :
  			IF NOT BlockedOpenControl THEN
                                IF  strKr.ISVALIDREF_cmdOn THEN strKr.CmdOn := TRUE;
  				IF strKr.ISVALIDREF_cmdOff THEN strKr.CmdOff := FALSE; END_IF;
  			ELSIF  strKr.ISVALIDREF_cmdOff THEN strKr.CmdOff := FALSE;  END_IF;
  			errorCMDTimer(IN := false);

  			_commandErrorTimer := true;
  			strKr.lastCmdIsOn := true;
                                END_IF;
  	(*cmd_close*) 2 :
  			IF strKr.ISVALIDREF_cmdOff THEN strKr.CmdOff := TRUE;
  				IF strKr.ISVALIDREF_cmdOn THEN strKr.CmdOn := FALSE; END_IF;
  			ELSIF strKr.ISVALIDREF_cmdOn THEN strKr.CmdOn := FALSE; END_IF;
  			errorCMDTimer(IN := false);

  			_commandErrorTimer := true;
  			strKr.lastCmdIsOn := false;
  	(*cmd_reset*) 3 :   IF (strKr.ISVALIDREF_statOn) OR (strKr.ISVALIDREF_statOff) THEN
  			strKr.CmdOn := FALSE;
  			strKr.CmdOff := FALSE;
                                lastCmd := 0;
  			_commandErrorTimer := false;
  			strKr.lastCmdIsOn := false;
                                END_IF;

  	END_CASE;
  	source_for_Status := source;
  	cmd_for_Status := cmd;
  	command_error_for_Status := 0;
  END_IF;
  lastCmd := cmd;

  errorCMDTimer(In := _commandErrorTimer, PT :=T#90s);

  continueHoldCommandTimer(IN:=(strKr.onStatus = _statusDualInput.STATUS_ON) OR
  (strKr.onStatus = _statusDualInput.STATUS_OFF), PT:=strKr.continueHoldCommand);

  (* ---- алгоритм  для команды ВКЛючить ---- *)
  IF (strKr.onStatus = _statusDualInput.STATUS_ON) and strKr.lastCmdIsOn  then
  	IF strKr.ISVALIDREF_cmdOn AND strKr.ISVALIDREF_cmdOff then
            IF continueHoldCommandTimer.Q THEN
            strKr.cmdOn := false; END_IF;
            END_IF;
  	 errorCMDTimer(In := false);
  	 _commandErrorTimer := false;
  	 cmd_for_Status := 0;
  	 source_for_Status := 0;
  END_IF;

  (* ---- off ---- *)
  IF (strKr.onStatus = _statusDualInput.STATUS_OFF) and  (NOT strKr.lastCmdIsOn) then
  	IF strKr.ISVALIDREF_cmdOn AND strKr.ISVALIDREF_cmdOff then
            IF continueHoldCommandTimer.Q THEN
            strKr.cmdOff := false; END_IF;
            END_IF;
  	 errorCMDTimer(In := false);
  	 _commandErrorTimer := false;
  	 cmd_for_Status := 0;
  	 source_for_Status := 0;
  END_IF;

  (* ---- ошибка исполнения команды ---- *)
  if errorCMDTimer.Q and (cmd_for_Status <> 0) then
  	command_error_for_Status :=  cmd_for_Status;
  	_commandErrorTimer := false;
  	strKr.CmdOn := false;
  	strKr.CmdOff := false;
  	(*lastCmd := 0;*)
  END_IF;

  (* ---- сброс ошибки команды ---- *)
  strKr.CommandFault := command_error_for_Status <> 0;
  _errorReset(IN := command_error_for_Status <> 0, PT := T#5S);
  IF _errorReset.Q THEN
  	cmd_for_Status := 0;
  	source_for_Status := 0;
  	command_error_for_Status := 0;

  END_IF;

  outputsSets(in := (strKr.ISVALIDREF_cmdOn and strKr.cmdOn ) OR (strKr.ISVALIDREF_cmdOff and strKr.cmdOff), PT := T#2S);
  	IF NOT outputsSets.Q THEN
  		strKr.So := inSo._inversed AND inSo.reliability AND strKr.ISVALIDREF_inSo;
  		strKr.Sz := inSz._inversed AND inSz.reliability AND strKr.ISVALIDREF_inSz;
  	END_IF;

  cmdOn := strKr.cmdOn;
  cmdOff:= strKr.cmdOff;

  (* ---- формирование зашифрованного статуса для АРМа ---- *)
  strKr.status := shl(BYTE_TO_DWORD(source_for_Status), 29)
  		OR shl(BYTE_TO_DWORD(cmd_for_Status), 26)
  		OR shl(BYTE_TO_DWORD(command_error_for_Status), 23)
  		OR shl(bool_to_DWORD(strKr.sdvig), 22)
  		OR shl(bool_to_DWORD(strKr.OpcCommandsDisabled), 21)
                      OR shl(bool_to_DWORD(strKr.Dp), 14)
                      OR shl(BOOL_TO_DWORD(strKr.Sz), 13)
  		OR shl(BOOL_TO_DWORD(strKr.So), 12)
  		OR shl(BOOL_TO_DWORD(strKr.ErrorBlock), 11)
  		OR shl(BOOL_TO_DWORD(strKr.ErrorPowerOff), 10)
  		OR shl(BOOL_TO_DWORD(strKr.Manual), 8)
  		OR shl(BOOL_TO_DWORD(strKr.Auto), 7)
  		OR shl(BOOL_TO_DWORD(strKr.Distance), 6)
  		OR shl(BOOL_TO_DWORD(strKr.Local), 5)
  		OR shl(BOOL_TO_DWORD(strKr.Ns), 4)
                  	OR shl(BOOL_TO_DWORD(strKr.Accident ),3)
  		OR BYTE_TO_DWORD(strKr.onStatus);
END_FUNCTION_BLOCK

FUNCTION_BLOCK fb_OilPump
  VAR_INPUT
    statOn : BOOL;
    statOff : BOOL;
    statOn_reliability : BOOL;
    statOff_reliability : BOOL;
  END_VAR
  VAR_IN_OUT
    StrSw : struct_OilPump;
  END_VAR
  VAR_INPUT
    inNs : TYPE_ReliableBit;
    inAccident : TYPE_ReliableBit;
    inLocal : TYPE_ReliableBit;
    inDistance : TYPE_ReliableBit;
    inBreakCmdOn : TYPE_ReliableBit;
    inBreakCmdOff : TYPE_ReliableBit;
  END_VAR
  VAR
    onInit : BOOL := FALSE;
    _statOn : BOOL;
    _statOff : BOOL;
    getSdvig : BOOL;
    lastOnStatus : BYTE;
    cmd : BYTE;
    source : BYTE;
    lastCmd : BYTE;
    source_for_Status : BYTE;
    cmd_for_Status : BYTE;
    command_error_for_Status : BYTE;
    _sunpackerCommand : fb_sunpackerCommand;
    _statusDualInput : TYPE_statusDualInput;
    _commandDualInput : TYPE_commandDualInput;
    _commandErrorTimer : BOOL;
    resetErrorTimer : BOOL;
    _changWithoutCommand : BOOL;
    errorCMDTimer : TON;
    sdvigReset : TON;
    _errorReset : TON;
    outputsSets : TOF;
  END_VAR
  VAR_IN_OUT
    cmdOn : BOOL;
    cmdOff : BOOL;
  END_VAR

  IF NOT onInit THEN
  IF StrSw.ISVALIDREF_cmdOn XOR StrSw.ISVALIDREF_cmdOff THEN
  	IF 	StrSw.ISVALIDREF_cmdOn THEN
  		lastCmd:= 2; (*baseCmdOff*)
  	ELSE
  		lastCmd:= 1; (*baseCmdOn*)
  	END_IF;
  END_IF;
  onInit:=TRUE;
  END_IF;

  (* ---- Если управление с ВУ заблокировано, то в ИМ передаем команду из алгоритма ---- *)
  IF StrSw.inOpcCommandsDisabled THEN
  	StrSw.inCommand := StrSw.inCommand_Alg;
  ELSE (* иначе передаем команду с АРМа*)
  	StrSw.inCommand := StrSw.inCommand_ARM;
  END_IF;

  (* ---- Формирование состояния механизма ---- *)

  IF (StrSw.ISVALIDREF_statOn) OR (StrSw.ISVALIDREF_statOff) THEN
  	IF (StrSw.ISVALIDREF_statOn) AND (StrSw.ISVALIDREF_statOff) THEN
  	StrSw.reliability:= statOn_reliability AND statOff_reliability;
  		_statOn  := statOn;
  		_statOff := statOff;
  	ELSIF (StrSw.ISVALIDREF_statOn) THEN
                       StrSw.reliability:= statOn_reliability;
  		_statOn  := statOn;
  		_statOff := NOT statOn;
  	ELSIF (StrSw.ISVALIDREF_statOff) THEN
  		 StrSw.reliability:= statOff_reliability;
  		_statOn  := NOT statOff;
  		_statOff :=statOff;
  	END_IF;

  	IF StrSw.reliability THEN
  		IF _statOn AND NOT _statOff 		THEN 	StrSw.onStatus := _statusDualInput.STATUS_ON;
  		ELSIF _statOff AND NOT _statOn 	THEN 	StrSw.onStatus := _statusDualInput.Status_OFF;
  		ELSIF NOT _statOn AND NOT _statOff 	THEN 	StrSw.onStatus := _statusDualInput.STATUS_TRANSITIONAL;
  		ELSE					StrSw.onStatus := _statusDualInput.STATUS_ERROR;
                      END_IF;

  	ELSE
  		StrSw.onStatus := _statusDualInput.STATUS_NOTDEFINED;

  	END_IF;
  ELSE
  	CASE BYTE_TO_INT(lastCmd) OF
  		(*baseCmdOn*) 1: StrSw.onStatus  := _statusDualInput.STATUS_ON;
  		(*baseCmdOff*) 2: StrSw.onStatus  := _statusDualInput.STATUS_OFF;

  	ELSE
  		 StrSw.onStatus := _statusDualInput.STATUS_NOTDEFINED;

  	END_CASE;
  END_IF;

  StrSw.Accident := inAccident.value AND inAccident.reliability;
  StrSw.Ns := inNs.value AND inNs.reliability;
  StrSw.Local := inLocal.value AND inLocal.reliability;
  StrSw.Distance := inDistance.value AND inDistance.reliability;
  StrSw.OpcCommandsDisabled := StrSw.inOpcCommandsDisabled;

  StrSw.Blocked:=StrSw.Accident OR StrSw.Local OR StrSw.breakCmdOn OR StrSw.breakCmdOff OR StrSw.inBlocked;

  StrSw.Rezervny:=NOT StrSw.Osnovnoy;

  (* ---- Формирование признака сдвига ---- *)

  getSdvig := FALSE;
  IF (StrSw.ISVALIDREF_cmdOn OR StrSw.ISVALIDREF_cmdOff) AND NOT StrSw.Local THEN
  	IF NOT (StrSw.CmdOn OR StrSw.CmdOff) THEN
                       IF (lastOnStatus <> StrSw.onStatus AND
  		(StrSw.onStatus <> _statusDualInput.STATUS_NOTDEFINED AND
                       StrSw.onStatus <> _statusDualInput.STATUS_ERROR)     AND
  		(lastOnStatus <> _statusDualInput.STATUS_NOTDEFINED   AND
                       lastOnStatus <> _statusDualInput.STATUS_ERROR))
                      THEN
  			getSdvig   := TRUE;
  		END_IF;
  	END_IF;
  END_IF;

  IF getSdvig THEN StrSw.sdvig:= TRUE; END_IF;

  sdvigReset(IN:=StrSw.sdvig, PT:=T#15S);

  IF sdvigReset.Q THEN StrSw.sdvig:=FALSE; END_IF;

  lastOnStatus := StrSw.onStatus;

  (* ---- Распаковка команды ---- *)
  _sunpackerCommand(command := StrSw.inCommand);
  	cmd := _sunpackerCommand.cmd;
  	source := _sunpackerCommand.source;

  (* ---- Обработка команды ---- *)
  IF cmd <> 0 AND lastCmd <> cmd and (((NOT StrSw.opcCommandsDisabled) AND source > 0) OR source = 0) then
  	CASE BYTE_TO_INT(cmd) OF
  	(*cmd_on*) 1 :
  			IF  StrSw.ISVALIDREF_cmdOn THEN StrSw.CmdOn := TRUE;
  				IF StrSw.ISVALIDREF_cmdOff THEN StrSw.CmdOff := FALSE; END_IF;
  			ELSIF  StrSw.ISVALIDREF_cmdOff THEN StrSw.CmdOff := FALSE;  END_IF;
  			errorCMDTimer(IN := false);
  			_commandErrorTimer := true;
  			StrSw.lastCmdIsOn := true;
  	(*cmd_off*) 2 :
  			IF StrSw.ISVALIDREF_cmdOff THEN StrSw.CmdOff := TRUE;
  				IF StrSw.ISVALIDREF_cmdOn THEN StrSw.CmdOn := FALSE; END_IF;
  			ELSIF StrSw.ISVALIDREF_cmdOn THEN StrSw.CmdOn := FALSE; END_IF;
  			errorCMDTimer(IN := false);

  			_commandErrorTimer := true;
  			StrSw.lastCmdIsOn := false;
  	(*cmd_reset*) 3 :    IF StrSw.ISVALIDREF_statOn OR StrSw.ISVALIDREF_statOff THEN
  			StrSw.CmdOn := FALSE;
  			StrSw.CmdOff := FALSE;
                                lastCmd := 0;
  			_commandErrorTimer := false;
  			StrSw.lastCmdIsOn := false;
                                 END_IF;
  	END_CASE;
  	source_for_Status := source;
  	cmd_for_Status := cmd;
  	command_error_for_Status := 0;
  END_IF;

  lastCmd := cmd;
  errorCMDTimer(In := _commandErrorTimer, PT :=T#10s);

  (* ---- алгоритм  для команды ВКЛючить ---- *)
  IF (StrSw.onStatus = _statusDualInput.STATUS_ON) and StrSw.lastCmdIsOn then
  	IF StrSw.ISVALIDREF_cmdOn AND StrSw.ISVALIDREF_cmdOff then  StrSw.cmdOn := false; END_IF;

  	 errorCMDTimer(In := false);
  	 _commandErrorTimer := false;
  	 cmd_for_Status := 0;
  	 source_for_Status := 0;
  END_IF;

  (* ---- off ---- *)
  IF (StrSw.onStatus = _statusDualInput.STATUS_OFF) and (NOT StrSw.lastCmdIsOn) then
  	IF StrSw.ISVALIDREF_cmdOn AND StrSw.ISVALIDREF_cmdOff then  StrSw.cmdOff := false; END_IF;

  	 errorCMDTimer(In := false);
  	 _commandErrorTimer := false;
  	 cmd_for_Status := 0;
  	 source_for_Status := 0;
  END_IF;

  (* ---- ошибка исполнения команды ---- *)
  if errorCMDTimer.Q and (cmd_for_Status <> 0) then
  	command_error_for_Status :=  cmd_for_Status;
  	_commandErrorTimer := false;
  	StrSw.CmdOn := false;
  	StrSw.CmdOff := false;
  	lastCmd := 0;
  end_if;

  (* ---- сброс ошибки команды ---- *)
  StrSw.CommandFault := command_error_for_Status <> 0;
  _errorReset(IN := command_error_for_Status <> 0, PT := T#5S);
  IF _errorReset.Q THEN
  	cmd_for_Status := 0;
  	source_for_Status := 0;
  	command_error_for_Status := 0;
  END_IF;

  outputsSets(in := (StrSw.ISVALIDREF_cmdOn and StrSw.cmdOn ) OR (StrSw.ISVALIDREF_cmdOff and StrSw.cmdOff), PT := T#2S);
  	IF NOT outputsSets.Q THEN
  		StrSw.BreakCmdOn := inBreakCmdOn._inversed AND inBreakCmdOn.reliability AND StrSw.ISVALIDREF_inBreakCmdOn;
  		StrSw.BreakCmdOff := inBreakCmdOff._inversed AND inBreakCmdOff.reliability AND StrSw.ISVALIDREF_inBreakCmdOff;
  	END_IF;

  cmdOn := StrSw.cmdOn;
  cmdOff:= StrSw.cmdOff;

  (* ---- формирование зашифрованного статуса для АРМа ---- *)
  StrSw.status := shl(BYTE_TO_DWORD(source_for_Status), 29)
  		OR shl(BYTE_TO_DWORD(cmd_for_Status), 26)
  		OR shl(BYTE_TO_DWORD(command_error_for_Status), 23)
  		OR shl(bool_to_DWORD(StrSw.sdvig), 22)
  		OR shl(bool_to_DWORD(StrSw.OpcCommandsDisabled), 21)
                      OR shl(bool_to_DWORD(StrSw.lastCmdIsOn), 14)
                      OR shl(BOOL_TO_DWORD(StrSw.BreakCmdOff), 13)
  		OR shl(BOOL_TO_DWORD(StrSw.BreakCmdOn), 12)
  		OR shl(BOOL_TO_DWORD(StrSw.Distance), 6)
  		OR shl(BOOL_TO_DWORD(StrSw.Local), 5)
  		OR shl(BOOL_TO_DWORD(StrSw.Ns), 4)
                  	OR shl(BOOL_TO_DWORD(StrSw.Accident ),3)
  		OR BYTE_TO_DWORD(StrSw.onStatus);
END_FUNCTION_BLOCK

FUNCTION_BLOCK fb_Switch
  VAR_INPUT
    statOn : BOOL;
    statOff : BOOL;
    statOn_reliability : BOOL;
    statOff_reliability : BOOL;
  END_VAR
  VAR_IN_OUT
    StrSw : struct_Switch;
  END_VAR
  VAR_INPUT
    inNs : TYPE_ReliableBit;
    inAccident : TYPE_ReliableBit;
    inAuto : TYPE_ReliableBit;
    inManual : TYPE_ReliableBit;
    inLocal : TYPE_ReliableBit;
    inDistance : TYPE_ReliableBit;
    inErrorPowerOff : TYPE_ReliableBit;
    inErrorBlock : TYPE_ReliableBit;
    inBreakCmdOn : TYPE_ReliableBit;
    inBreakCmdOff : TYPE_ReliableBit;
  END_VAR
  VAR
    onInit : BOOL := FALSE;
    _statOn : BOOL;
    _statOff : BOOL;
    lastOnStatus : BYTE;
    cmd : BYTE;
    source : BYTE;
    lastCmd : BYTE;
    source_for_Status : BYTE;
    cmd_for_Status : BYTE;
    command_error_for_Status : BYTE;
    _sunpackerCommand : fb_sunpackerCommand;
    _statusDualInput : TYPE_statusDualInput;
    _commandDualInput : TYPE_commandDualInput;
    _commandErrorTimer : BOOL;
    resetErrorTimer : BOOL;
    getSdvig : BOOL;
    _changWithoutCommand : BOOL;
    errorCMDTimer : TON;
    sdvigReset : TON;
    _errorReset : TON;
    outputsSets : TOF;
  END_VAR
  VAR_IN_OUT
    cmdOn : BOOL;
    cmdOff : BOOL;
  END_VAR

  IF NOT onInit THEN
  IF StrSw.ISVALIDREF_cmdOn XOR StrSw.ISVALIDREF_cmdOff THEN
  	IF 	StrSw.ISVALIDREF_cmdOn THEN
  		lastCmd:= 2; (*baseCmdOff*)
  	ELSE
  		lastCmd:= 1; (*baseCmdOn*)
  	END_IF;
  END_IF;
  onInit:=TRUE;
  END_IF;

  (* ---- Если управление с ВУ заблокировано, то в ИМ передаем команду из алгоритма ---- *)
  IF StrSw.inOpcCommandsDisabled THEN
  	StrSw.inCommand := StrSw.inCommand_Alg;
  ELSE (* иначе передаем команду с АРМа*)
  	StrSw.inCommand := StrSw.inCommand_ARM;
  END_IF;

  (* ---- Формирование состояния механизма ---- *)

  IF (StrSw.ISVALIDREF_statOn) OR (StrSw.ISVALIDREF_statOff) THEN
  	IF (StrSw.ISVALIDREF_statOn) AND (StrSw.ISVALIDREF_statOff) THEN
  	StrSw.reliability:= statOn_reliability AND statOff_reliability;
  		_statOn  := statOn;
  		_statOff := statOff;
  	ELSIF (StrSw.ISVALIDREF_statOn) THEN
                       StrSw.reliability:= statOn_reliability;
  		_statOn  := statOn;
  		_statOff := NOT statOn;
  	ELSIF (StrSw.ISVALIDREF_statOff) THEN
  		 StrSw.reliability:= statOff_reliability;
  		_statOn  := NOT statOff;
  		_statOff :=statOff;
  	END_IF;

  	IF StrSw.reliability THEN
  		IF _statOn AND NOT _statOff 		THEN 	StrSw.onStatus := _statusDualInput.STATUS_ON;
  		ELSIF _statOff AND NOT _statOn 	THEN 	StrSw.onStatus := _statusDualInput.Status_OFF;
  		ELSIF NOT _statOn AND NOT _statOff 	THEN 	StrSw.onStatus := _statusDualInput.STATUS_TRANSITIONAL;
  		ELSE					StrSw.onStatus := _statusDualInput.STATUS_ERROR;
                      END_IF;

  	ELSE
  		StrSw.onStatus := _statusDualInput.STATUS_NOTDEFINED;

  	END_IF;
  ELSE
  	CASE BYTE_TO_INT(lastCmd) OF
  		(*baseCmdOn*) 1: StrSw.onStatus  := _statusDualInput.STATUS_ON;
  		(*baseCmdOff*) 2: StrSw.onStatus  := _statusDualInput.STATUS_OFF;

  	ELSE
  		 StrSw.onStatus := _statusDualInput.STATUS_NOTDEFINED;

  	END_CASE;
  END_IF;

  StrSw.Accident := inAccident.value AND inAccident.reliability;
  StrSw.Ns := inNs.value AND inNs.reliability;
  StrSw.Auto := inAuto.value AND inAuto.reliability;
  StrSw.Manual := inManual.value AND inManual.reliability;
  StrSw.Local := inLocal.value AND inLocal.reliability;
  StrSw.Distance := inDistance.value AND inDistance.reliability;
  StrSw.ErrorPowerOff := inErrorPowerOff.value AND inErrorPowerOff.reliability;
  StrSw.ErrorBlock := inErrorBlock.value AND inErrorBlock.reliability;
  StrSw.OpcCommandsDisabled := StrSw.inOpcCommandsDisabled;

  (* ---- Формирование признака сдвига ---- *)
  getSdvig := FALSE;
  IF (StrSw.ISVALIDREF_cmdOn OR StrSw.ISVALIDREF_cmdOff) AND NOT StrSw.Local THEN
  	IF NOT (StrSw.CmdOn OR StrSw.CmdOff) THEN
                       IF (lastOnStatus <> StrSw.onStatus AND
  		(StrSw.onStatus <> _statusDualInput.STATUS_NOTDEFINED AND
                       StrSw.onStatus <> _statusDualInput.STATUS_ERROR)     AND
  		(lastOnStatus <> _statusDualInput.STATUS_NOTDEFINED   AND
                       lastOnStatus <> _statusDualInput.STATUS_ERROR))
                      THEN
  			getSdvig   := TRUE;
  		END_IF;
  	END_IF;
  END_IF;
